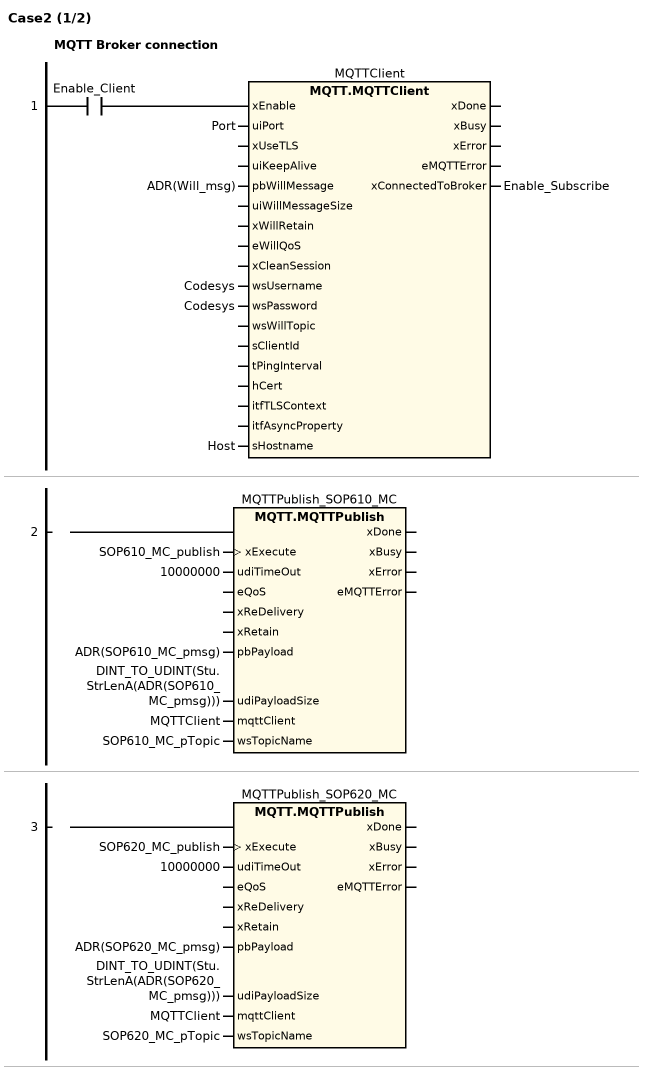
// NETWORK 1: MQTT Broker connection
MQTTClient(
    xEnable := Enable_Client,
    uiPort := Port,
    pbWillMessage := ADR(Will_msg),
    wsUsername := Codesys,
    wsPassword := Codesys,
    sHostname := Host,
    xConnectedToBroker => Enable_Subscribe); // MQTT.MQTTClient

// NETWORK 2
_rt1(CLK := SOP610_MC_publish);
MQTTPublish_SOP610_MC(
    xExecute := _rt1.Q,
    udiTimeOut := 10000000,
    pbPayload := ADR(SOP610_MC_pmsg),
    udiPayloadSize := DINT_TO_UDINT(Stu.StrLenA(ADR(SOP610_MC_pmsg))),
    mqttClient := MQTTClient,
    wsTopicName := SOP610_MC_pTopic); // MQTT.MQTTPublish

// NETWORK 3
_rt2(CLK := SOP620_MC_publish);
MQTTPublish_SOP620_MC(
    xExecute := _rt2.Q,
    udiTimeOut := 10000000,
    pbPayload := ADR(SOP620_MC_pmsg),
    udiPayloadSize := DINT_TO_UDINT(Stu.StrLenA(ADR(SOP620_MC_pmsg))),
    mqttClient := MQTTClient,
    wsTopicName := SOP620_MC_pTopic); // MQTT.MQTTPublish

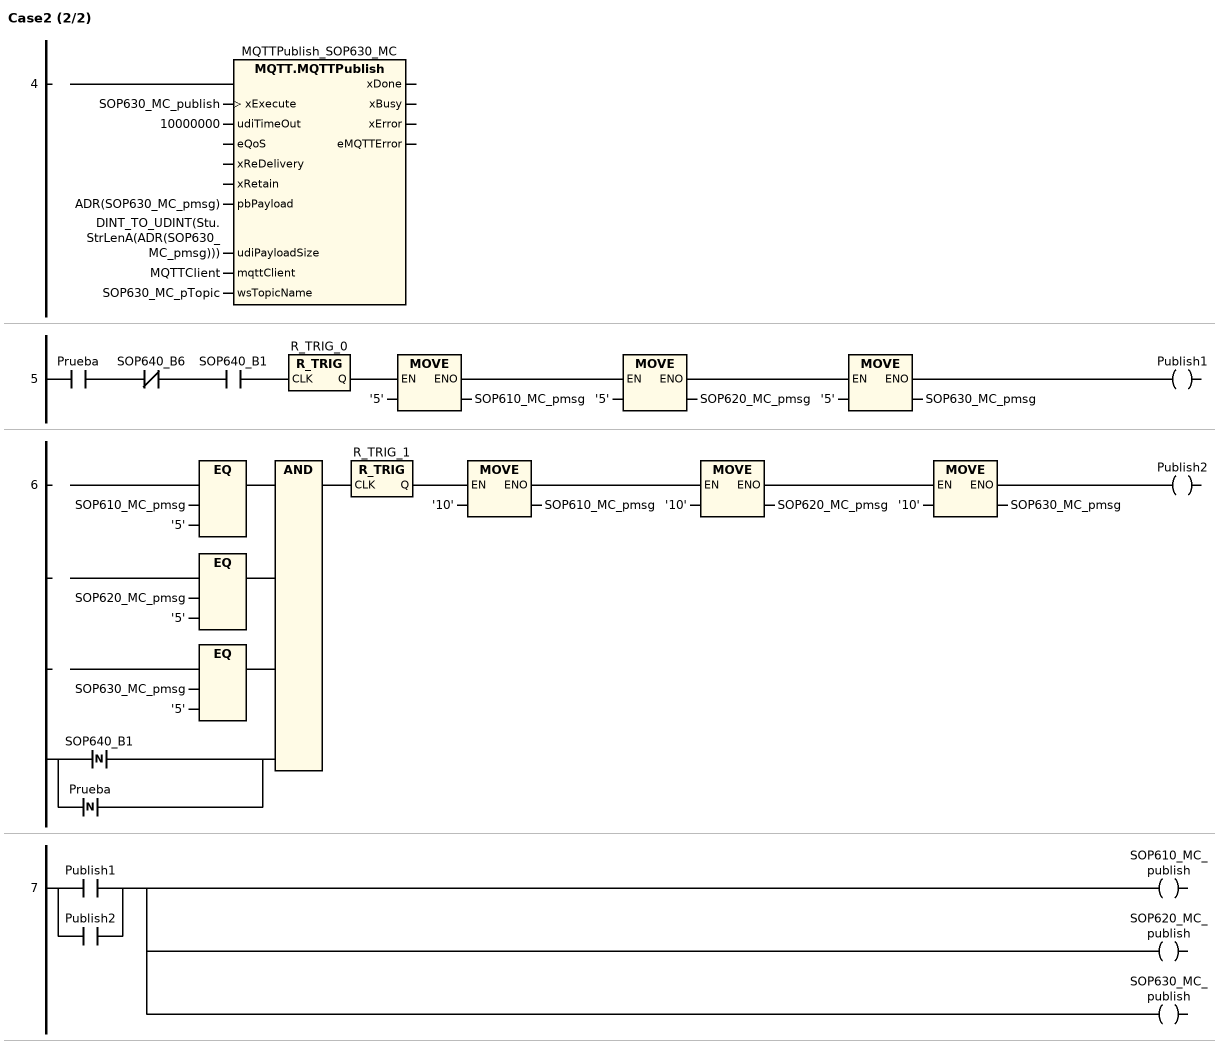
// NETWORK 4
_rt3(CLK := SOP630_MC_publish);
MQTTPublish_SOP630_MC(
    xExecute := _rt3.Q,
    udiTimeOut := 10000000,
    pbPayload := ADR(SOP630_MC_pmsg),
    udiPayloadSize := DINT_TO_UDINT(Stu.StrLenA(ADR(SOP630_MC_pmsg))),
    mqttClient := MQTTClient,
    wsTopicName := SOP630_MC_pTopic); // MQTT.MQTTPublish

// NETWORK 5
R_TRIG_0(CLK := Prueba AND NOT SOP640_B6 AND SOP640_B1); // R_TRIG
_w1 := R_TRIG_0.Q;
IF _w1 THEN SOP610_MC_pmsg := '5'; END_IF
IF _w1 THEN SOP620_MC_pmsg := '5'; END_IF
IF _w1 THEN SOP630_MC_pmsg := '5'; END_IF
Publish1 := _w1;

// NETWORK 6
_ft1(CLK := SOP640_B1);
_ft2(CLK := Prueba);
R_TRIG_1(CLK := SOP610_MC_pmsg = '5' AND SOP620_MC_pmsg = '5' AND SOP630_MC_pmsg = '5' AND (_ft1.Q OR _ft2.Q)); // R_TRIG
_w2 := R_TRIG_1.Q;
IF _w2 THEN SOP610_MC_pmsg := '10'; END_IF
IF _w2 THEN SOP620_MC_pmsg := '10'; END_IF
IF _w2 THEN SOP630_MC_pmsg := '10'; END_IF
Publish2 := _w2;

// NETWORK 7
_w3 := Publish1 OR Publish2;
SOP610_MC_publish := _w3;
SOP620_MC_publish := _w3;
SOP630_MC_publish := _w3;

END_PROGRAM

// Device/Application/Cases/Cases3_4_5
PROGRAM Cases3_4_5
VAR
	MQTTClient: MQTT.MQTTClient; 										// MQTTClient FB
	Port: UINT := 1883; 												// Port
	Will_msg: STRING(1024) := ''; 										// Message if there is disconnection
	Host: STRING(255) := '192.168.1.123'; 								// Broker IP 192.168.1.123 Simumatik
	Codesys: WSTRING(1024) := "codesys";								// Username and password "Codesys"
	Enable_Client: BOOL := TRUE; 										// Establishes connecting with the MQTT broker
	Enable_Subscribe: BOOL;												// Enables subscription
	
	MQTTPublish_SOP610_MC: MQTT.MQTTPublish;								// MQTTPublish FB
	SOP610_MC_publish: BOOL;
	SOP610_MC_pmsg: STRING(1024);
	SOP610_MC_pTopic: WSTRING(1024) := "OP60/SOP610_MC";	
	MQTTPublish_SOP620_MC: MQTT.MQTTPublish;								// MQTTPublish FB
	SOP620_MC_publish: BOOL;
	SOP620_MC_pmsg: STRING(1024);
	SOP620_MC_pTopic: WSTRING(1024) := "OP60/SOP620_MC";
	MQTTPublish_SOP630_MC: MQTT.MQTTPublish;								// MQTTPublish FB
	SOP630_MC_publish: BOOL;
	SOP630_MC_pmsg: STRING(1024);
	SOP630_MC_pTopic: WSTRING(1024) := "OP60/SOP630_MC";
	MQTTPublish_SOP640_MC: MQTT.MQTTPublish;								// MQTTPublish FB
	SOP640_MC_publish: BOOL;
	SOP640_MC_pmsg: STRING(1024);
	SOP640_MC_pTopic: WSTRING(1024) := "OP60/SOP640_MC";
	MQTTPublish_SOP650_MC: MQTT.MQTTPublish;								// MQTTPublish FB
	SOP650_MC_publish: BOOL;
	SOP650_MC_pmsg: STRING(1024);
	SOP650_MC_pTopic: WSTRING(1024) := "OP60/SOP650_MC";
	MQTTPublish_SOP660_MC: MQTT.MQTTPublish;								// MQTTPublish FB
	SOP660_MC_publish: BOOL;
	SOP660_MC_pmsg: STRING(1024);
	SOP660_MC_pTopic: WSTRING(1024) := "OP60/SOP660_MC";
	MQTTPublish_SOP670_MC: MQTT.MQTTPublish;								// MQTTPublish FB
	SOP670_MC_publish: BOOL;
	SOP670_MC_pmsg: STRING(1024);
	SOP670_MC_pTopic: WSTRING(1024) := "OP60/SOP670_MC";
	MQTTPublish_SOP680_MC: MQTT.MQTTPublish;								// MQTTPublish FB
	SOP680_MC_publish: BOOL;
	SOP680_MC_pmsg: STRING(1024);
	SOP680_MC_pTopic: WSTRING(1024) := "OP60/SOP680_MC";
	
	MQTTSubscribe_MC: MQTT.MQTTSubscribe;
	Subscribe_Topic: WSTRING(1024) := "OP60/MC";
	Subscribe_msg: STRING(1024);
	Subscribe_msg_received: BOOL;
	
	R_TRIG_0: R_TRIG;
	R_TRIG_1: R_TRIG;
	R_TRIG_2: R_TRIG;
	R_TRIG_3: R_TRIG;
	R_TRIG_4: R_TRIG;
	R_TRIG_5: R_TRIG;
	R_TRIG_6: R_TRIG;
	R_TRIG_7: R_TRIG;
	R_TRIG_8: R_TRIG;
	Iniciate_publish: BOOL;
	TON_0: TON;
END_VAR
VAR_INPUT
	iSOP610_MC: BOOL;
	iSOP620_MC: BOOL;
	iSOP630_MC: BOOL;
	iSOP640_MC: BOOL;
	iSOP650_MC: BOOL;
	iSOP660_MC: BOOL;
	iSOP670_MC: BOOL;
	iSOP680_MC: BOOL;
END_VAR
VAR // added by the converter: edge detectors and wires of the graphical bodies
    _rt1, _rt2, _rt3, _rt4, _rt5, _rt6, _rt7, _rt8 : R_TRIG;
    _w1, _w2, _w3, _w4, _w5, _w6, _w7, _w8, _w9 : BOOL;
END_VAR

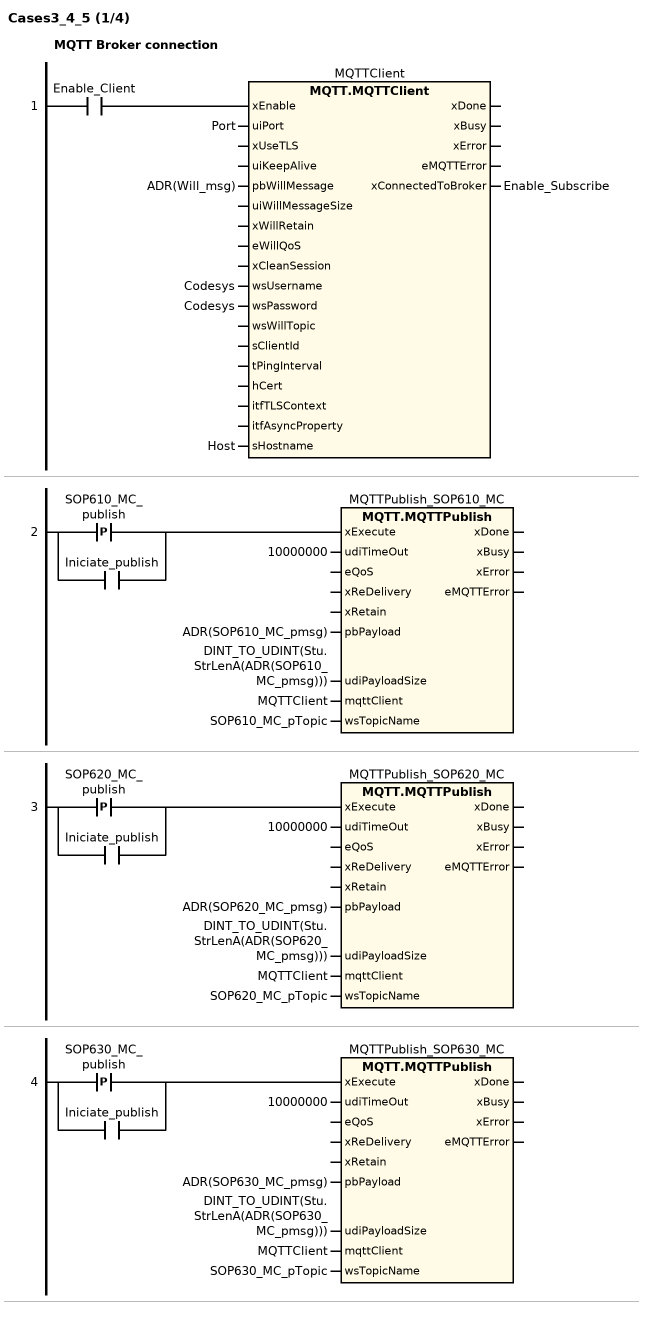
// NETWORK 1: MQTT Broker connection
MQTTClient(
    xEnable := Enable_Client,
    uiPort := Port,
    pbWillMessage := ADR(Will_msg),
    wsUsername := Codesys,
    wsPassword := Codesys,
    sHostname := Host,
    xConnectedToBroker => Enable_Subscribe); // MQTT.MQTTClient

// NETWORK 2
_rt1(CLK := SOP610_MC_publish);
MQTTPublish_SOP610_MC(
    xExecute := _rt1.Q OR Iniciate_publish,
    udiTimeOut := 10000000,
    pbPayload := ADR(SOP610_MC_pmsg),
    udiPayloadSize := DINT_TO_UDINT(Stu.StrLenA(ADR(SOP610_MC_pmsg))),
    mqttClient := MQTTClient,
    wsTopicName := SOP610_MC_pTopic); // MQTT.MQTTPublish

// NETWORK 3
_rt2(CLK := SOP620_MC_publish);
MQTTPublish_SOP620_MC(
    xExecute := _rt2.Q OR Iniciate_publish,
    udiTimeOut := 10000000,
    pbPayload := ADR(SOP620_MC_pmsg),
    udiPayloadSize := DINT_TO_UDINT(Stu.StrLenA(ADR(SOP620_MC_pmsg))),
    mqttClient := MQTTClient,
    wsTopicName := SOP620_MC_pTopic); // MQTT.MQTTPublish

// NETWORK 4
_rt3(CLK := SOP630_MC_publish);
MQTTPublish_SOP630_MC(
    xExecute := _rt3.Q OR Iniciate_publish,
    udiTimeOut := 10000000,
    pbPayload := ADR(SOP630_MC_pmsg),
    udiPayloadSize := DINT_TO_UDINT(Stu.StrLenA(ADR(SOP630_MC_pmsg))),
    mqttClient := MQTTClient,
    wsTopicName := SOP630_MC_pTopic); // MQTT.MQTTPublish

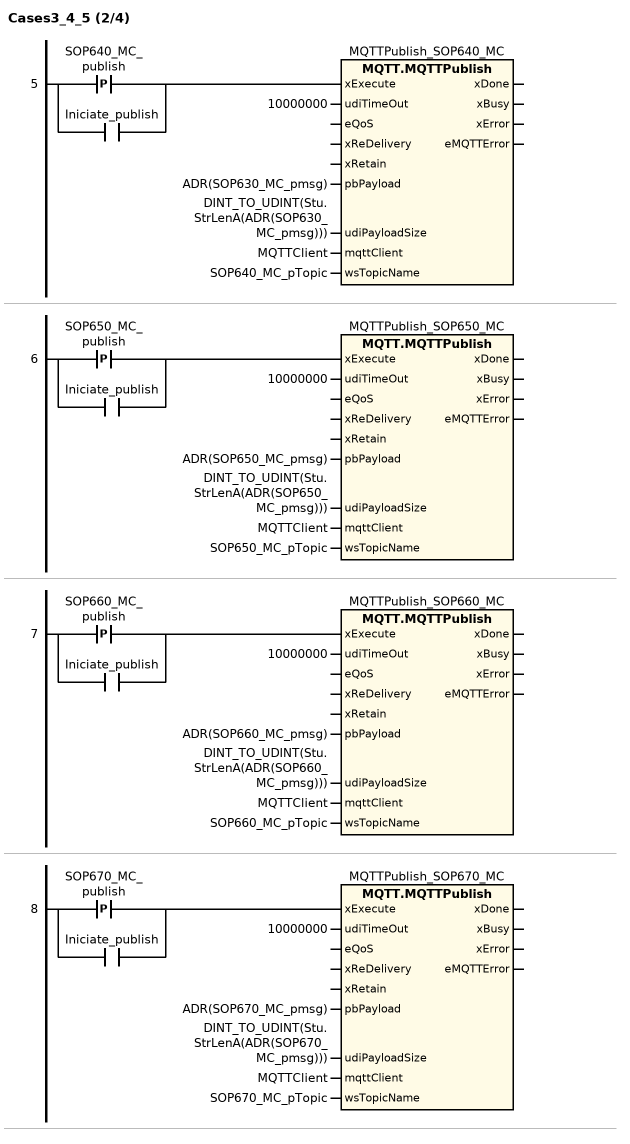
// NETWORK 5
_rt4(CLK := SOP640_MC_publish);
MQTTPublish_SOP640_MC(
    xExecute := _rt4.Q OR Iniciate_publish,
    udiTimeOut := 10000000,
    pbPayload := ADR(SOP630_MC_pmsg),
    udiPayloadSize := DINT_TO_UDINT(Stu.StrLenA(ADR(SOP630_MC_pmsg))),
    mqttClient := MQTTClient,
    wsTopicName := SOP640_MC_pTopic); // MQTT.MQTTPublish

// NETWORK 6
_rt5(CLK := SOP650_MC_publish);
MQTTPublish_SOP650_MC(
    xExecute := _rt5.Q OR Iniciate_publish,
    udiTimeOut := 10000000,
    pbPayload := ADR(SOP650_MC_pmsg),
    udiPayloadSize := DINT_TO_UDINT(Stu.StrLenA(ADR(SOP650_MC_pmsg))),
    mqttClient := MQTTClient,
    wsTopicName := SOP650_MC_pTopic); // MQTT.MQTTPublish

// NETWORK 7
_rt6(CLK := SOP660_MC_publish);
MQTTPublish_SOP660_MC(
    xExecute := _rt6.Q OR Iniciate_publish,
    udiTimeOut := 10000000,
    pbPayload := ADR(SOP660_MC_pmsg),
    udiPayloadSize := DINT_TO_UDINT(Stu.StrLenA(ADR(SOP660_MC_pmsg))),
    mqttClient := MQTTClient,
    wsTopicName := SOP660_MC_pTopic); // MQTT.MQTTPublish

// NETWORK 8
_rt7(CLK := SOP670_MC_publish);
MQTTPublish_SOP670_MC(
    xExecute := _rt7.Q OR Iniciate_publish,
    udiTimeOut := 10000000,
    pbPayload := ADR(SOP670_MC_pmsg),
    udiPayloadSize := DINT_TO_UDINT(Stu.StrLenA(ADR(SOP670_MC_pmsg))),
    mqttClient := MQTTClient,
    wsTopicName := SOP670_MC_pTopic); // MQTT.MQTTPublish

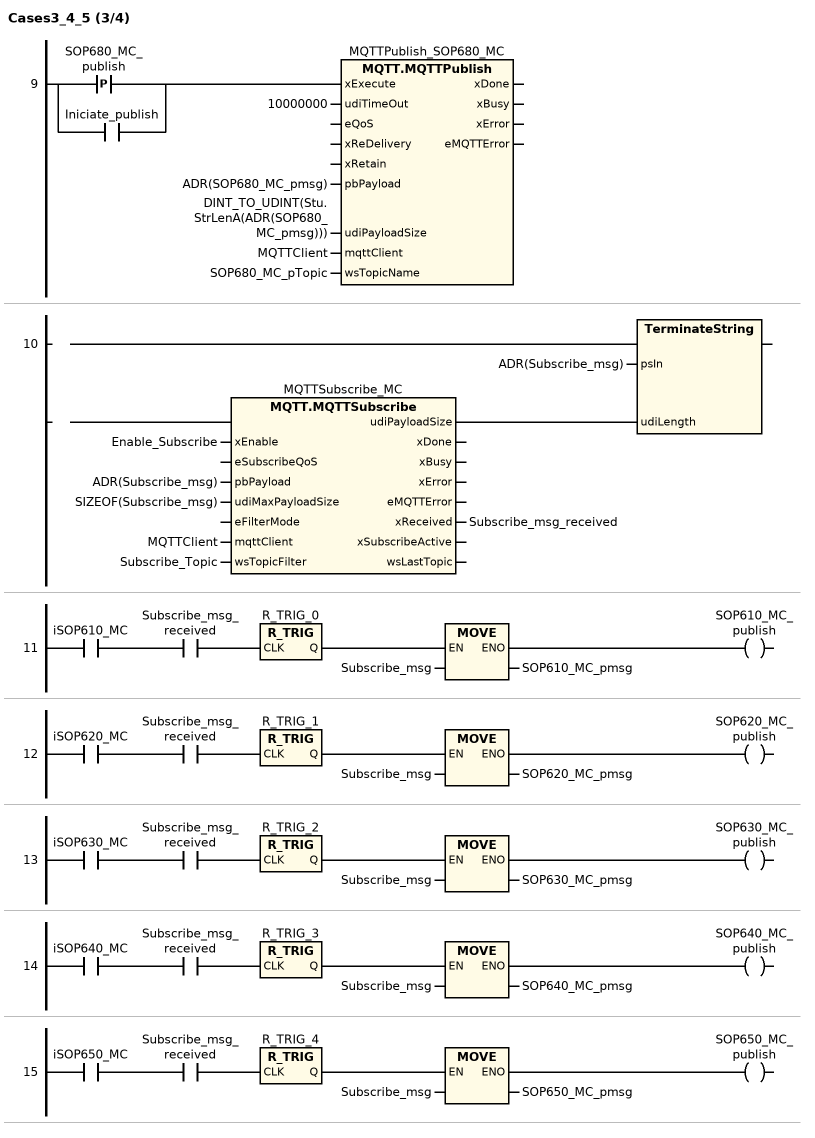
// NETWORK 9
_rt8(CLK := SOP680_MC_publish);
MQTTPublish_SOP680_MC(
    xExecute := _rt8.Q OR Iniciate_publish,
    udiTimeOut := 10000000,
    pbPayload := ADR(SOP680_MC_pmsg),
    udiPayloadSize := DINT_TO_UDINT(Stu.StrLenA(ADR(SOP680_MC_pmsg))),
    mqttClient := MQTTClient,
    wsTopicName := SOP680_MC_pTopic); // MQTT.MQTTPublish

// NETWORK 10
MQTTSubscribe_MC(
    xEnable := Enable_Subscribe,
    pbPayload := ADR(Subscribe_msg),
    udiMaxPayloadSize := SIZEOF(Subscribe_msg),
    mqttClient := MQTTClient,
    wsTopicFilter := Subscribe_Topic,
    xReceived => Subscribe_msg_received); // MQTT.MQTTSubscribe
TerminateString(psIn := ADR(Subscribe_msg), udiLength := MQTTSubscribe_MC.udiPayloadSize);

// NETWORK 11
R_TRIG_0(CLK := iSOP610_MC AND Subscribe_msg_received); // R_TRIG
_w1 := R_TRIG_0.Q;
IF _w1 THEN SOP610_MC_pmsg := Subscribe_msg; END_IF
SOP610_MC_publish := _w1;

// NETWORK 12
R_TRIG_1(CLK := iSOP620_MC AND Subscribe_msg_received); // R_TRIG
_w2 := R_TRIG_1.Q;
IF _w2 THEN SOP620_MC_pmsg := Subscribe_msg; END_IF
SOP620_MC_publish := _w2;

// NETWORK 13
R_TRIG_2(CLK := iSOP630_MC AND Subscribe_msg_received); // R_TRIG
_w3 := R_TRIG_2.Q;
IF _w3 THEN SOP630_MC_pmsg := Subscribe_msg; END_IF
SOP630_MC_publish := _w3;

// NETWORK 14
R_TRIG_3(CLK := iSOP640_MC AND Subscribe_msg_received); // R_TRIG
_w4 := R_TRIG_3.Q;
IF _w4 THEN SOP640_MC_pmsg := Subscribe_msg; END_IF
SOP640_MC_publish := _w4;

// NETWORK 15
R_TRIG_4(CLK := iSOP650_MC AND Subscribe_msg_received); // R_TRIG
_w5 := R_TRIG_4.Q;
IF _w5 THEN SOP650_MC_pmsg := Subscribe_msg; END_IF
SOP650_MC_publish := _w5;

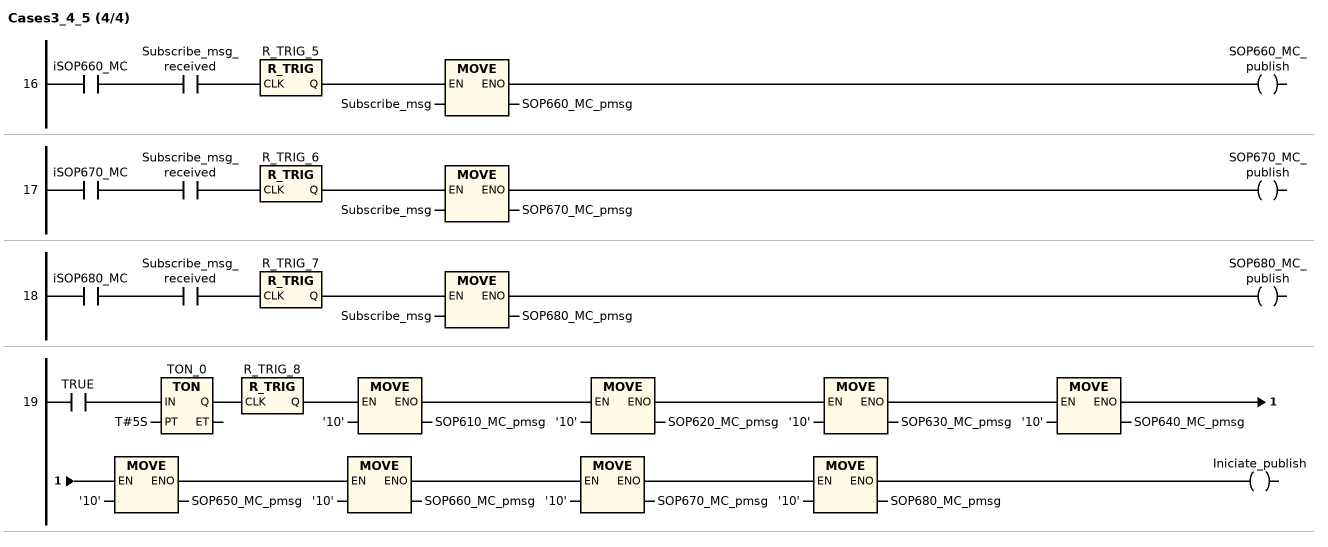
// NETWORK 16
R_TRIG_5(CLK := iSOP660_MC AND Subscribe_msg_received); // R_TRIG
_w6 := R_TRIG_5.Q;
IF _w6 THEN SOP660_MC_pmsg := Subscribe_msg; END_IF
SOP660_MC_publish := _w6;

// NETWORK 17
R_TRIG_6(CLK := iSOP670_MC AND Subscribe_msg_received); // R_TRIG
_w7 := R_TRIG_6.Q;
IF _w7 THEN SOP670_MC_pmsg := Subscribe_msg; END_IF
SOP670_MC_publish := _w7;

// NETWORK 18
R_TRIG_7(CLK := iSOP680_MC AND Subscribe_msg_received); // R_TRIG
_w8 := R_TRIG_7.Q;
IF _w8 THEN SOP680_MC_pmsg := Subscribe_msg; END_IF
SOP680_MC_publish := _w8;

// NETWORK 19
TON_0(IN := TRUE, PT := T#5S); // TON
R_TRIG_8(CLK := TON_0.Q); // R_TRIG
_w9 := R_TRIG_8.Q;
IF _w9 THEN SOP610_MC_pmsg := '10'; END_IF
IF _w9 THEN SOP620_MC_pmsg := '10'; END_IF
IF _w9 THEN SOP630_MC_pmsg := '10'; END_IF
IF _w9 THEN SOP640_MC_pmsg := '10'; END_IF
IF _w9 THEN SOP650_MC_pmsg := '10'; END_IF
IF _w9 THEN SOP660_MC_pmsg := '10'; END_IF
IF _w9 THEN SOP670_MC_pmsg := '10'; END_IF
IF _w9 THEN SOP680_MC_pmsg := '10'; END_IF
Iniciate_publish := _w9;

END_PROGRAM

// Device/Application/MQTTSub
PROGRAM MQTTSub
VAR
	//Define Client
	MQTTCLient5 : MQTT.MQTTClient;		
	MQTTReady: BOOL;								
	Enable_Client : BOOL := TRUE;										
	Port : UINT := 1883;
	Will_msg: STRING(1024) := ''; 										// Message if there is disconnection
	Host: STRING(255) := '192.168.1.123'; 								// Broker IP 192.168.1.123 Simumatik
	Codesys: WSTRING(1024) := "codesys";
	
	// Define Subscriber
	MQTTSubscriber: MQTT.MQTTSubscribe;
	Enable_Subscribe: BOOL;
	Received_messages: ARRAY [1..3] OF STRING(1024) := ['', '', ''];	// Received messages
	New_message: ARRAY [1..3] OF BOOL;									// This is done to avoid errors
	Topics: ARRAY [1..3] OF WSTRING(1024) := ["Subscriber1","Subscriber2","Subscriber3"];
	
	i: DINT := 1;
	Delay: TON;
	DelayTime: TIME;
END_VAR

MQTTClient5(xEnable:=Enable_Client, uiPort:=Port, pbWillMessage:=ADR(Will_msg), wsUsername:=Codesys, wsPassword:=Codesys, sHostname:=Host, xConnectedToBroker => MQTTReady);  // Define Client

IF MQTTReady THEN
	MQTTSubscriber(xEnable:= TRUE, pbPayload:= ADR(Received_messages[i]), udiMaxPayloadSize:= SIZEOF(Received_messages[i]), mqttClient:= MQTTClient5, wsTopicFilter:= Topics[i], xReceived => New_message[i]);
	Delay(IN:=TRUE, PT:=T#100MS, ET => DelayTime);
	IF NOT(Delay.Q) THEN
		RETURN;
	END_IF
	Delay(IN:=FALSE);
	MQTTSubscriber(xEnable:= FALSE, pbPayload:= ADR(Received_messages[i]), udiMaxPayloadSize:= SIZEOF(Received_messages[i]), mqttClient:= MQTTClient5, wsTopicFilter:= Topics[i], xReceived => New_message[i]);
END_IF

IF i = (UPPER_BOUND(Received_messages,1)) THEN
	i := LOWER_BOUND(Received_messages,1)-1;
END_IF
i := i+1;

END_PROGRAM

// Device/Application/FBs/EraseSeconds
FUNCTION EraseSeconds : STRING // Returns TIME STRING in HH:MM:SS to HH:MM format 
VAR_INPUT
	iTime_hh_mm_ss: STRING;
END_VAR
VAR
END_VAR

EraseSeconds := LEFT(iTime_hh_mm_ss,5);

END_FUNCTION

// Device/Application/Pruebas
PROGRAM Pruebas
VAR

	Output: SysFile.RTS_IEC_HANDLE;
	TON_0: TON;
	TimerON: BOOL;
	TimerON_0: TIME;
	Salida: __XWORD;
	pbyBuffer: POINTER TO BYTE := 4096;
	ulSize: __XWORD := 4096;
	pResult: POINTER TO SysFile.RTS_IEC_RESULT;
	szFile: REFERENCE TO STRING;
END_VAR

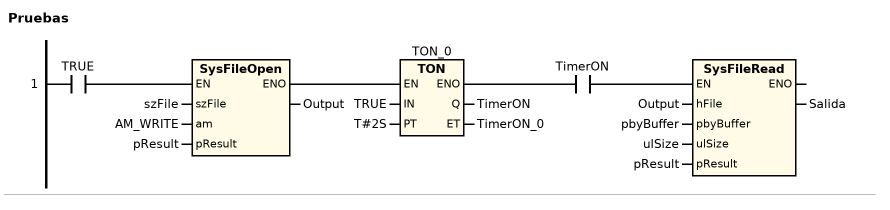
// NETWORK 1
Output := SysFileOpen(szFile := szFile, am := AM_WRITE, pResult := pResult);
TON_0(IN := TRUE, PT := T#2S, Q => TimerON, ET => TimerON_0); // TON
IF TRUE AND TimerON THEN
    Salida := SysFileRead(hFile := Output, pbyBuffer := pbyBuffer, ulSize := ulSize, pResult := pResult);
END_IF

END_PROGRAM

// Device/Application/MQTTPub
PROGRAM MQTTPub
VAR
	//Define Client
	MQTTCLient4 : MQTT.MQTTClient;										
	Enable_Client : BOOL := TRUE;										
	Port : UINT := 1883;
	Will_msg: STRING(1024) := ''; 										// Message if there is disconnection
	Host: STRING(255) := '192.168.1.123'; 								// Broker IP 192.168.1.123 Simumatik
	Codesys: WSTRING(1024) := "codesys";
	Enable_Publish: BOOL;												// Rising edge activates Publisher FB
	
	//Define Publisher
	MQTTPublisher: MQTT.MQTTPublish;
	Topics: ARRAY [1..3] OF WSTRING(1024) := ["Publish","Publish2","Publish3"];	// All the topics
	Publish_msg: ARRAY [1..3] OF STRING(1024);			// Messages to publish
	Publish_last_msg: ARRAY [1..3] OF STRING(1024);		// Last messages to publish

	i : DINT := 1; 		//index
	Delay: TON;			// Timer to delay
END_VAR

MQTTClient4(xEnable:=Enable_Client, uiPort:=Port, pbWillMessage:=ADR(Will_msg), wsUsername:=Codesys, wsPassword:=Codesys, sHostname:=Host,);  // Define Client

// Publish the messages that have change
IF NOT (Publish_msg[i] = Publish_last_msg[i]) THEN
	Enable_Publish:= TRUE;
	MQTTPublisher(xExecute:=Enable_Publish, udiTimeOut:=1000000, pbPayload:=ADR(Publish_msg[i]), udiPayloadSize:=DINT_TO_UDINT(Stu.StrLenA(ADR(Publish_msg[i]))), mqttclient:=MQTTClient4, wsTopicName:=Topics[i]);
	// Delay 50miliseconds;
	Delay(IN:=TRUE, PT:=T#50MS);
	IF NOT(Delay.Q) THEN
   		RETURN;
	END_IF
	Delay(IN:=FALSE);
	Enable_Publish:= FALSE;
	MQTTPublisher(xExecute:=FALSE, udiTimeOut:=1000000, pbPayload:=ADR(Publish_msg[i]), udiPayloadSize:=DINT_TO_UDINT(Stu.StrLenA(ADR(Publish_msg[i]))), mqttclient:=MQTTClient4, wsTopicName:=Topics[i]);
	// To avoid missing messages
	//MQTTPublisher(xExecute:=TRUE, udiTimeOut:=1000000, pbPayload:=ADR(Publish_msg[i]), udiPayloadSize:=DINT_TO_UDINT(Stu.StrLenA(ADR(Publish_msg[i]))), mqttclient:=MQTTClient4, wsTopicName:=Topics[i]);
	//MQTTPublisher(xExecute:=FALSE, udiTimeOut:=1000000, pbPayload:=ADR(Publish_msg[i]), udiPayloadSize:=DINT_TO_UDINT(Stu.StrLenA(ADR(Publish_msg[i]))), mqttclient:=MQTTClient4, wsTopicName:=Topics[i]);
	
	Publish_last_msg[i] := Publish_msg[i];
	
END_IF

// IF Enable_Publish = TRUE THEN
// 	// Delay 50miliseconds;
// 	Delay(IN:=TRUE, PT:=T#50MS);
// 	IF NOT(Delay.Q) THEN
//    		RETURN;
// 	END_IF
// 	Delay(IN:=FALSE);
// 	Enable_Publish:= FALSE;
// 	MQTTPublisher(xExecute:=Enable_Publish);
// END_IF


// Control the index
IF i = (UPPER_BOUND(Publish_msg,1)) THEN
	i := LOWER_BOUND(Publish_msg,1)-1;
END_IF
i := i+1;

END_PROGRAM

// Device/Application/Production
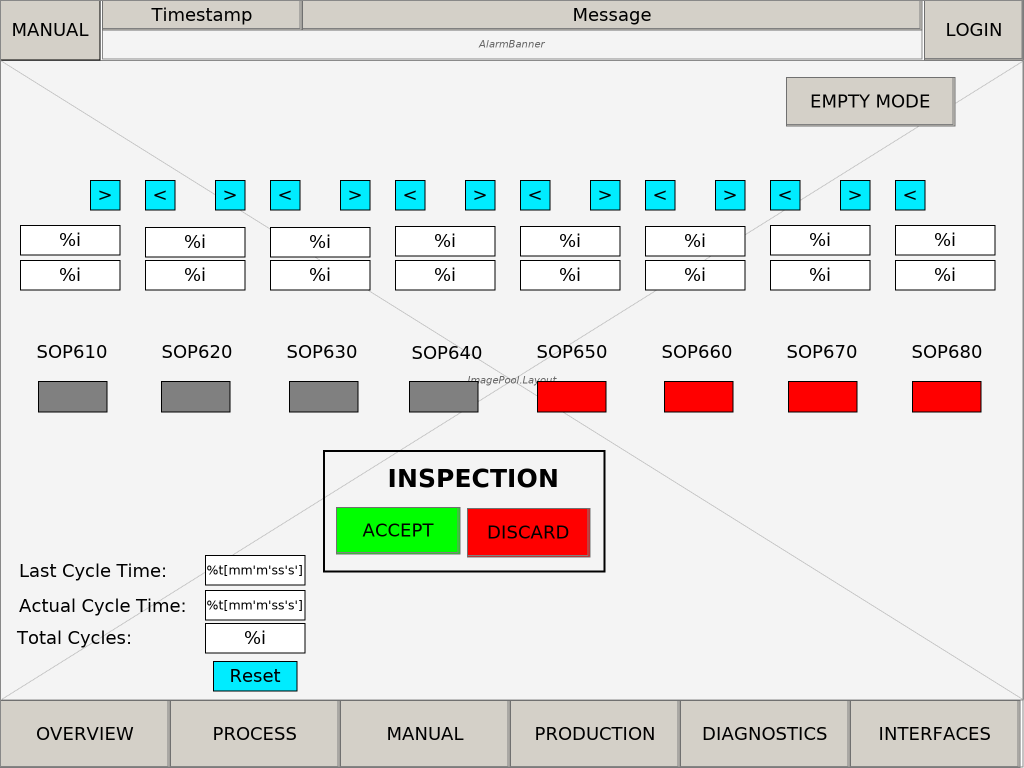
VISUALIZATION Production  // 1024x768, background image ImagePool.Layout
    Image (0,60 1024x640), image: ImagePool.Layout
    Rectangle (0,0 100x60), "AUTO"
    Rectangle (0,0 100x60), "MANUAL", invisible if: OP60_Auto
    AlarmBanner (102,29 820x30)
        p1521930926: __All
        p1663851261: __All
    Button (924,0 100x60), "LOGIN"
    Button (102,0 200x30), "Timestamp"
    Button (302,0 620x30), "Message"
    Label (145,337 104x30), "SOP620"
    Label (20,337 104x30), "SOP610"
    Label (270,337 104x30), "SOP630"
    Label (395,338 104x30), "SOP640"
    Label (520,337 104x30), "SOP650"
    Label (645,337 104x30), "SOP660"
    Label (895,337 104x30), "SOP680"
    Label (770,337 104x30), "SOP670"
    Rectangle (20,260 100x30), "%i", text variable: SOP610_PD.ProductNr
    Rectangle (20,225 100x30), "%i", text variable: SOP610_PD.IDNumber
    Rectangle (145,227 100x30), "%i", text variable: SOP620_PD.IDNumber
    Rectangle (145,260 100x30), "%i", text variable: SOP620_PD.ProductNr
    Rectangle (270,227 100x30), "%i", text variable: SOP630_PD.IDNumber
    Rectangle (270,260 100x30), "%i", text variable: SOP630_PD.ProductNr
    Rectangle (395,226 100x30), "%i", text variable: SOP640_PD.IDNumber
    Rectangle (395,260 100x30), "%i", text variable: SOP640_PD.ProductNr
    Rectangle (520,226 100x30), "%i", text variable: SOP650_PD.IDNumber
    Rectangle (520,260 100x30), "%i", text variable: SOP650_PD.ProductNr
    Rectangle (645,226 100x30), "%i", text variable: SOP660_PD.IDNumber
    Rectangle (645,260 100x30), "%i", text variable: SOP660_PD.ProductNr
    Rectangle (770,225 100x30), "%i", text variable: SOP670_PD.IDNumber
    Rectangle (770,260 100x30), "%i", text variable: SOP670_PD.ProductNr
    Rectangle (895,225 100x30), "%i", text variable: SOP680_PD.IDNumber
    Rectangle (895,260 100x30), "%i", text variable: SOP680_PD.ProductNr
    Group (323,450 282x122), invisible if: not HMI_SOP640_Inspecting
        Rectangle (0,0 282x122)
        Button (13,57 124x47), "ACCEPT"
            tap HMI_SOP640_Accept
        Label (39,13 223x30), "INSPECTION"
        Button (144,58 123x49), "DISCARD"
            tap HMI_SOP640_Discard
    Group (0,700 1020x68)
        Button (0,0 170x68), "OVERVIEW"
            toggle OP60_Visu.CV_Overview
            OnMouseDown:  Assign=Overview, Type=Assignment
        Button (170,0 170x68), "PROCESS"
            toggle OP60_Visu.CV_Process
            OnMouseDown:  Assign=Process, Type=Assignment
        Button (340,0 170x68), "MANUAL"
            toggle OP60_Visu.CV_Manual_SOP610t630
            OnMouseDown:  Assign=Manual_SOP610t630, Type=Assignment
        Button (510,0 170x68), "PRODUCTION"
            toggle OP60_Visu.CV_Production
            OnMouseDown:  Assign=Production, Type=Assignment
        Button (680,0 170x68), "DIAGNOSTICS"
            toggle OP60_Visu.CV_Diagnostics
            OnMouseDown:  Assign=Diagnostics, Type=Assignment
        Button (850,0 170x68), "INTERFACES"
            toggle OP60_Visu.CV_Interfaces
            OnMouseDown:  Assign=Interfaces, Type=Assignment
    Rectangle (90,180 30x30), ">"
        tap HMI_SOP610_ManPDFwd
    Rectangle (215,180 30x30), ">"
        tap HMI_SOP620_ManPDFwd
    Rectangle (145,180 30x30), "<"
        tap HMI_SOP620_ManPDRev
    Rectangle (340,180 30x30), ">"
        tap HMI_SOP630_ManPDFwd
    Rectangle (270,180 30x30), "<"
        tap HMI_SOP630_ManPDRev
    Rectangle (465,180 30x30), ">"
        tap HMI_SOP640_ManPDFwd
    Rectangle (395,180 30x30), "<"
        tap HMI_SOP640_ManPDRev
    Rectangle (590,180 30x30), ">"
        tap HMI_SOP650_ManPDFwd
    Rectangle (520,180 30x30), "<"
        tap HMI_SOP650_ManPDRev
    Rectangle (715,180 30x30), ">"
        tap HMI_SOP660_ManPDFwd
    Rectangle (645,180 30x30), "<"
        tap HMI_SOP660_ManPDRev
    Rectangle (840,180 30x30), ">"
        tap HMI_SOP670_ManPDFwd
    Rectangle (770,180 30x30), "<"
        tap HMI_SOP670_ManPDRev
    Rectangle (895,180 30x30), "<"
        tap HMI_SOP680_ManPDRev
    Label (16,591 193x30), "Actual Cycle Time:"
    Label (14,623 193x30), "Total Cycles:"
    Rectangle (213,661 84x30), "Reset"
        tap HMI_TotalCyclesReset
    Rectangle (205,590 100x30), "%t[mm'm'ss's']", text variable: OP60_ActualCycleTime
    Rectangle (205,623 100x30), "%i", text variable: OP60_TotalCycles
    Button (786,77 169x49), "EMPTY MODE"
        toggle GVL.OP60_EmptyMode
    Group (38,381 943x31)
        Rectangle (371,0 69x31), invisible if: not STRING_TO_BOOL(SOP640_B1_msg)
        Rectangle (251,0 69x31), invisible if: not STRING_TO_BOOL(SOP630_B1_msg)
        Rectangle (123,0 69x31), invisible if: not STRING_TO_BOOL(SOP620_B1_msg)
        Rectangle (0,0 69x31), invisible if: not STRING_TO_BOOL(SOP610_B1_msg)
        Rectangle (499,0 69x31), invisible if: not STRING_TO_BOOL(SOP650_B1_msg)
            toggle SOP650_PD.Status.6
        Rectangle (626,0 69x31), invisible if: not STRING_TO_BOOL(SOP660_B1_msg)
            toggle SOP660_PD.Status.6
        Rectangle (750,0 69x31), invisible if: not STRING_TO_BOOL(SOP670_B1_msg)
            toggle SOP670_PD.Status.6
        Rectangle (874,0 69x31), invisible if: not STRING_TO_BOOL(SOP680_B1_msg)
            toggle SOP680_PD.Status.6
    Label (16,556 193x30), "Last Cycle Time:"
    Rectangle (205,555 100x30), "%t[mm'm'ss's']", text variable: OP60_LastCycleTime
END_VISUALIZATION

// /Diagnostics
VISUALIZATION Diagnostics  // 1024x768
END_VISUALIZATION

// Device/Application/Overview
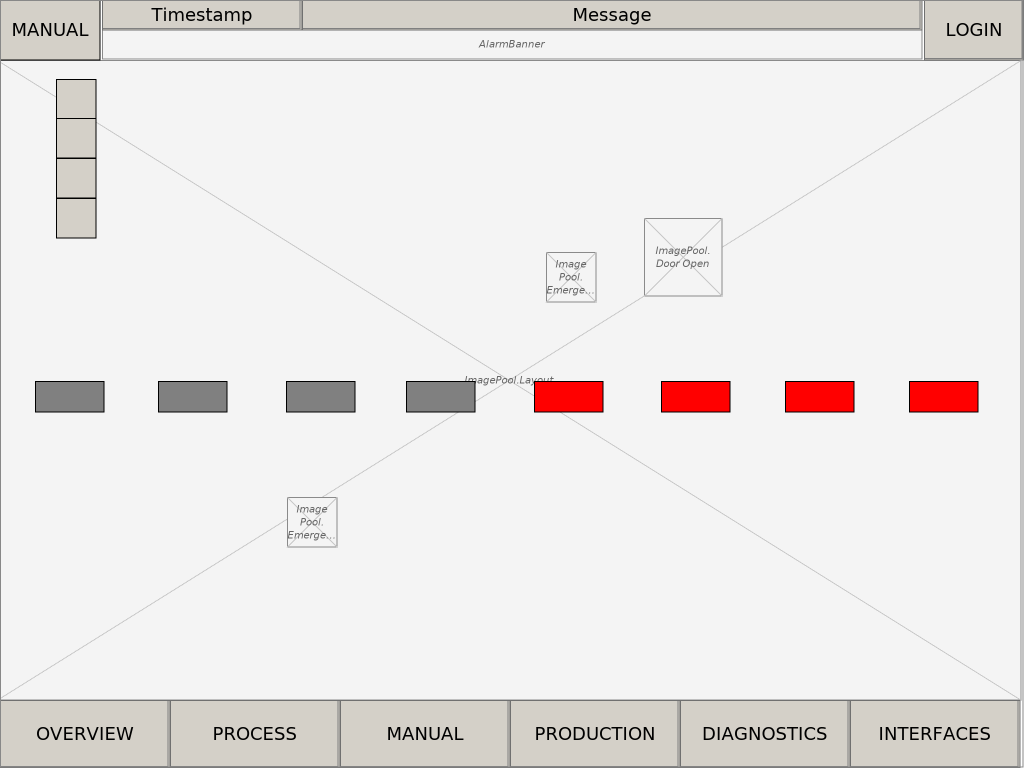
VISUALIZATION Overview  // 1024x768
    Image (-3,60 1024x640), image: ImagePool.Layout
    Rectangle (0,0 100x60), "AUTO"
    Rectangle (0,0 100x60), "MANUAL", invisible if: OP60_Auto
    AlarmBanner (102,29 820x30)
        p1521930926: __All
        p1663851261: __All
    Button (924,0 100x60), "LOGIN"
    Button (102,0 200x30), "Timestamp"
    Button (302,0 620x30), "Message"
    Group (56,79 40x159)
        Rectangle (0,0 40x40)
            toggle SOP600_H9
        Rectangle (0,39 40x40)
            toggle SOP600_H8
        Rectangle (0,79 40x40)
            toggle SOP600_H7
        Rectangle (0,119 40x40)
            toggle SOP600_H6
    Image (287,497 50x50), invisible if: SOP600_NS1, image: ImagePool.Emergency Stop
    Image (546,252 50x50), invisible if: SOP690_NS1, image: ImagePool.Emergency Stop
    Image (644,218 78x78), invisible if: SOP690_B1, image: ImagePool.Door Open
    Group (0,700 1020x68)
        Button (0,0 170x68), "OVERVIEW"
            toggle OP60_Visu.CV_Overview
            OnMouseDown:  Assign=Overview, Type=Assignment
        Button (170,0 170x68), "PROCESS"
            toggle OP60_Visu.CV_Process
            OnMouseDown:  Assign=Process, Type=Assignment
        Button (340,0 170x68), "MANUAL"
            toggle OP60_Visu.CV_Manual_SOP610t630
            OnMouseDown:  Assign=Manual_SOP610t630, Type=Assignment
        Button (510,0 170x68), "PRODUCTION"
            toggle OP60_Visu.CV_Production
            OnMouseDown:  Assign=Production, Type=Assignment
        Button (680,0 170x68), "DIAGNOSTICS"
            toggle OP60_Visu.CV_Diagnostics
            OnMouseDown:  Assign=Diagnostics, Type=Assignment
        Button (850,0 170x68), "INTERFACES"
            toggle OP60_Visu.CV_Interfaces
            OnMouseDown:  Assign=Interfaces, Type=Assignment
    Group (35,381 943x31)
        Rectangle (371,0 69x31), invisible if: not STRING_TO_BOOL(SOP640_B1_msg)
        Rectangle (251,0 69x31), invisible if: not STRING_TO_BOOL(SOP630_B1_msg)
        Rectangle (123,0 69x31), invisible if: not STRING_TO_BOOL(SOP620_B1_msg)
        Rectangle (0,0 69x31), invisible if: not STRING_TO_BOOL(SOP610_B1_msg)
        Rectangle (499,0 69x31), invisible if: not STRING_TO_BOOL(SOP650_B1_msg)
            toggle SOP650_PD.Status.6
        Rectangle (626,0 69x31), invisible if: not STRING_TO_BOOL(SOP660_B1_msg)
            toggle SOP660_PD.Status.6
        Rectangle (750,0 69x31), invisible if: not STRING_TO_BOOL(SOP670_B1_msg)
            toggle SOP670_PD.Status.6
        Rectangle (874,0 69x31), invisible if: not STRING_TO_BOOL(SOP680_B1_msg)
            toggle SOP680_PD.Status.6
END_VISUALIZATION

// Device/Application/Manual_SOP640
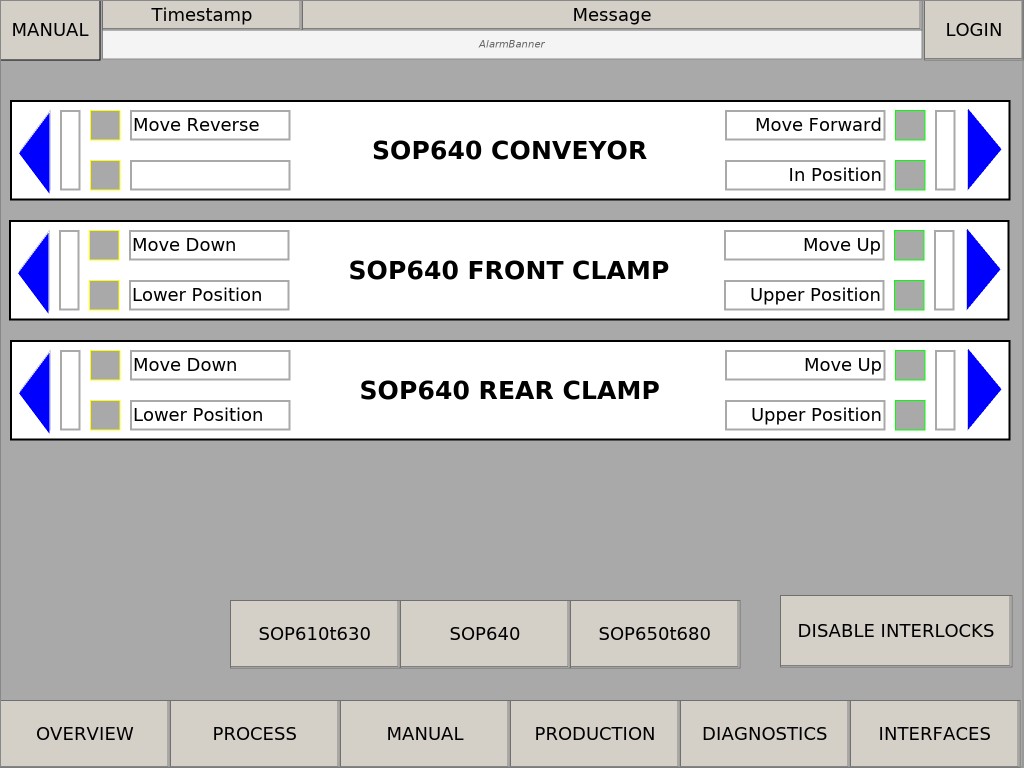
VISUALIZATION Manual_SOP640  // 1024x768
    Rectangle (0,0 100x60), "AUTO"
    Rectangle (0,0 100x60), "MANUAL", invisible if: OP60_Auto
    AlarmBanner (102,29 820x30)
        p1521930926: __All
        p1663851261: __All
    Button (924,0 100x60), "LOGIN"
    Button (102,0 200x30), "Timestamp"
    Button (302,0 620x30), "Message"
    Button (0,700 170x68), "OVERVIEW"
        toggle OP60_Visu.CV_Overview
        OnMouseDown:  Assign=Overview, Type=Assignment
    Button (170,700 170x68), "PROCESS"
        toggle OP60_Visu.CV_Process
        OnMouseDown:  Assign=Process, Type=Assignment
    Button (340,700 170x68), "MANUAL"
        toggle OP60_Visu.CV_Manual_SOP610t630
        OnMouseDown:  Assign=Manual_SOP610t630, Type=Assignment
    Button (510,700 170x68), "PRODUCTION"
        toggle OP60_Visu.CV_Production
        OnMouseDown:  Assign=Production, Type=Assignment
    Button (680,700 170x68), "DIAGNOSTICS"
        toggle OP60_Visu.CV_Diagnostics
        OnMouseDown:  Assign=Diagnostics, Type=Assignment
    Button (850,700 170x68), "INTERFACES"
        toggle OP60_Visu.CV_Interfaces
        OnMouseDown:  Assign=Interfaces, Type=Assignment
    Group (10,100 1000x100)
        Rectangle (0,0 1000x100), "SOP640 CONVEYOR"
        Polygon (10,50) (40,10) (40,90) (10,50) (10,50)
        Rectangle (50,10 20x80)
            toggle HMI_SOP640_ManMoveRev
        Polygon (990,50) (957,10) (957,90) (990,50) (990,50)
        Rectangle (925,10 20x80)
            toggle HMI_SOP640_ManMoveFwd
        Rectangle (715,10 160x30), "Move Forward"
        Rectangle (715,60 160x30), "In Position"
        Rectangle (120,10 160x30), "Move Reverse"
        Rectangle (120,60 160x30), invisible if: TRUE
        Rectangle (885,10 30x30)
            toggle SOP640_KM1
        Rectangle (80,60 30x30), invisible if: TRUE
        Rectangle (80,10 30x30)
            toggle SOP640_KM2
        Rectangle (885,60 30x30)
            toggle SOP640_B1
        Polygon (991,49) (958,9) (958,89) (991,49) (991,49), invisible if: not OP60_Manual
            tap HMI_SOP640_ManMoveFwd
        Polygon (9,53) (39,13) (39,93) (9,53) (9,53), invisible if: not OP60_Manual
            tap HMI_SOP640_ManMoveRev
    Group (9,220 1000x100)
        Rectangle (0,0 1000x100), "SOP640 FRONT CLAMP"
        Polygon (10,50) (40,10) (40,90) (10,50) (10,50)
        Rectangle (50,10 20x80)
            toggle HMI_SOP640_ManFrontDown
        Polygon (990,50) (957,10) (957,90) (990,50) (990,50)
        Rectangle (925,10 20x80)
            toggle HMI_SOP640_ManFrontUp
        Rectangle (715,10 160x30), "Move Up"
        Rectangle (715,60 160x30), "Upper Position"
        Rectangle (120,10 160x30), "Move Down"
        Rectangle (120,60 160x30), "Lower Position", invisible if: TRUE
        Rectangle (885,10 30x30)
            toggle SOP640_Y1
        Rectangle (80,60 30x30)
            toggle SOP640_B2
        Rectangle (80,10 30x30)
            toggle SOP640_Y2
        Rectangle (885,60 30x30)
            toggle SOP640_B3
        Polygon (991,49) (958,9) (958,89) (991,49) (991,49), invisible if: not OP60_Manual
            tap HMI_SOP640_ManFrontUp
        Polygon (9,53) (39,13) (39,93) (9,53) (9,53), invisible if: not OP60_Manual
            tap HMI_SOP640_ManFrontDown
    Group (230,600 510x68)
        Button (0,0 170x68), "SOP610t630"
            toggle OP60_Visu.CV_Manual_SOP610t630
            OnMouseDown:  Assign=Manual_SOP610t630, Type=Assignment
        Button (170,0 170x68), "SOP640"
            toggle OP60_Visu.CV_Manual_SOP640
            OnMouseDown:  Assign=Manual_SOP640, Type=Assignment
        Button (340,0 170x68), "SOP650t680"
            toggle OP60_Visu.CV_Manual_SOP650t680
            OnMouseDown:  Assign=Manual_SOP650t680, Type=Assignment
    Rectangle (10,340 1000x100), "SOP640 REAR CLAMP"
    Polygon (20,390) (50,350) (50,430) (20,390) (20,390)
    Rectangle (60,350 20x80)
        toggle HMI_SOP640_ManRearDown
    Polygon (1000,390) (967,350) (967,430) (1000,390) (1000,390)
    Rectangle (935,350 20x80)
        toggle HMI_SOP640_ManRearUp
    Rectangle (725,350 160x30), "Move Up"
    Rectangle (725,400 160x30), "Upper Position"
    Rectangle (130,350 160x30), "Move Down"
    Rectangle (130,400 160x30), "Lower Position", invisible if: TRUE
    Rectangle (895,350 30x30)
        toggle SOP640_Y3
    Rectangle (90,400 30x30)
        toggle SOP640_B4
    Rectangle (90,350 30x30)
        toggle SOP640_Y4
    Rectangle (895,400 30x30)
        toggle SOP640_B5
    Polygon (1001,389) (968,349) (968,429) (1001,389) (1001,389), invisible if: not OP60_Manual
        tap HMI_SOP640_ManRearUp
    Polygon (19,393) (49,353) (49,433) (19,393) (19,393), invisible if: not OP60_Manual
        tap HMI_SOP640_ManRearDown
    Button (780,595 232x72), "DISABLE INTERLOCKS", invisible if: not OP60_Manual
        toggle HMI_DisableInterlocks
END_VISUALIZATION

// Device/Application/Process
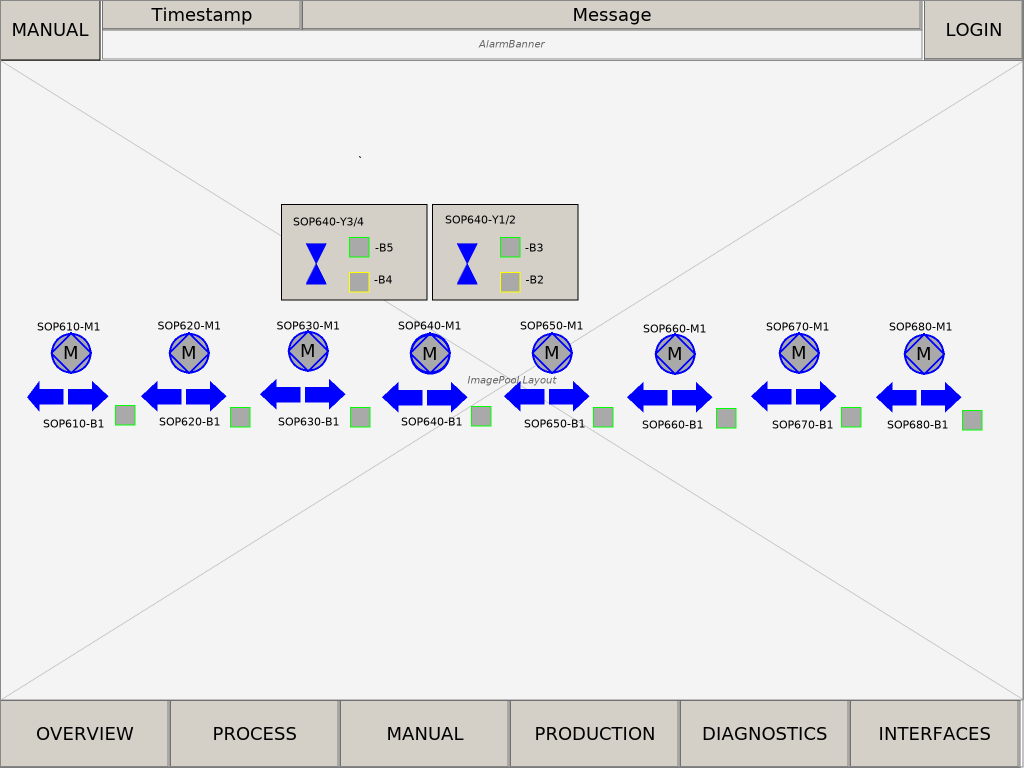
VISUALIZATION Process  // 1024x768
    Image (0,60 1024x640), image: ImagePool.Layout
    Rectangle (432,204 146x96)
    Rectangle (0,0 100x60), "AUTO"
    Rectangle (0,0 100x60), "MANUAL", invisible if: OP60_Auto
    AlarmBanner (102,29 820x30)
        p1521930926: __All
        p1663851261: __All
    Button (924,0 100x60), "LOGIN"
    Button (102,0 200x30), "Timestamp"
    Button (302,0 620x30), "Message"
    Rectangle (115,405 20x20)
        toggle SOP610_B1
    Label (22,409 104x30), "SOP610-B1"
    Ellipse (51,333 40x40), "M"
        toggle SOP610_Conveyor.oRunning
    Ellipse (51,333 40x40)
        toggle SOP610_Conveyor.oFaulted
    Polyline (51,353) (71,333) (91,353) (71,373) (51,353)
        toggle SOP610_Conveyor.oFaulted
    Rectangle (68,389 24x15), invisible if: not SOP610_Conveyor.oRunFwd and not SOP610_Conveyor.oFaulted
        toggle SOP610_Conveyor.oFaulted
    Polygon (92,388) (92,381) (108,396) (92,411) (92,403), invisible if: not SOP610_Conveyor.oRunFwd and not SOP610_Conveyor.oFaulted
        toggle SOP610_Conveyor.oFaulted
    Polygon (39,388) (39,381) (27,397) (39,411) (39,403), invisible if: not SOP610_Conveyor.oRunRev and not SOP610_Conveyor.oFaulted
        toggle SOP610_Conveyor.oFaulted
    Rectangle (39,389 24x15), invisible if: not SOP610_Conveyor.oRunRev and not SOP610_Conveyor.oFaulted
        toggle SOP610_Conveyor.oFaulted
    Label (138,407 104x30), "SOP620-B1"
    Label (257,407 104x30), "SOP630-B1"
    Label (366,407 132x30), "SOP640-B1"
    Label (503,409 104x30), "SOP650-B1"
    Label (621,410 104x30), "SOP660-B1"
    Label (866,410 104x30), "SOP680-B1"
    Label (751,410 104x30), "SOP670-B1"
    Rectangle (230,407 20x20)
        toggle SOP620_B1 p2164770859=TRUE
    Rectangle (350,407 20x20)
        toggle SOP630_B1
    Rectangle (471,406 20x20)
        toggle SOP640_B1
    Rectangle (593,407 20x20)
        toggle SOP650_B1
    Rectangle (716,408 20x20)
        toggle SOP660_B1
    Rectangle (841,407 20x20)
        toggle SOP670_B1
    Rectangle (962,410 20x20)
        toggle SOP680_B1
    Rectangle (186,389 24x15), invisible if: not SOP620_Conveyor.oRunFwd and not SOP620_Conveyor.oFaulted
        toggle SOP620_Conveyor.oFaulted
    Polygon (210,388) (210,381) (226,396) (210,411) (210,403), invisible if: not SOP620_Conveyor.oRunFwd and not SOP620_Conveyor.oFaulted
        toggle SOP620_Conveyor.oFaulted
    Ellipse (169,333 40x40), "M"
        toggle SOP620_Conveyor.oRunning
    Polygon (157,388) (157,381) (141,396) (157,411) (157,403), invisible if: not SOP620_Conveyor.oRunRev and not SOP620_Conveyor.oFaulted
        toggle SOP620_Conveyor.oFaulted
    Rectangle (157,389 24x15), invisible if: not SOP620_Conveyor.oRunRev and not SOP620_Conveyor.oFaulted
        toggle SOP620_Conveyor.oFaulted
    Rectangle (305,387 24x15), invisible if: not SOP630_Conveyor.oRunFwd and not SOP630_Conveyor.oFaulted
        toggle SOP630_Conveyor.oFaulted
    Polygon (329,386) (329,379) (345,394) (329,409) (329,401), invisible if: not SOP630_Conveyor.oRunFwd and not SOP630_Conveyor.oFaulted
        toggle SOP630_Conveyor.oFaulted
    Ellipse (288,331 40x40), "M"
        toggle SOP630_Conveyor.oRunning
    Polygon (276,386) (276,379) (260,394) (276,409) (276,401), invisible if: not SOP630_Conveyor.oRunRev and not SOP630_Conveyor.oFaulted
        toggle SOP630_Conveyor.oFaulted
    Rectangle (276,387 24x15), invisible if: not SOP630_Conveyor.oRunRev and not SOP630_Conveyor.oFaulted
        toggle SOP630_Conveyor.oFaulted
    Rectangle (427,390 24x15), invisible if: not SOP640_Conveyor.oRunFwd and not SOP640_Conveyor.oFaulted
        toggle SOP640_Conveyor.oFaulted
    Polygon (451,389) (451,382) (467,397) (451,412) (451,404), invisible if: not SOP640_Conveyor.oRunFwd and not SOP640_Conveyor.oFaulted
        toggle SOP640_Conveyor.oFaulted
    Ellipse (410,334 40x40), "M"
        toggle SOP640_Conveyor.oRunning
    Polygon (398,389) (398,382) (382,397) (398,412) (398,404), invisible if: not SOP640_Conveyor.oRunRev and not SOP640_Conveyor.oFaulted
        toggle SOP640_Conveyor.oFaulted
    Rectangle (398,390 24x15), invisible if: not SOP640_Conveyor.oRunRev and not SOP640_Conveyor.oFaulted
        toggle SOP640_Conveyor.oFaulted
    Rectangle (549,389 24x15), invisible if: not SOP650_Conveyor.oRunFwd and not SOP650_Conveyor.oFaulted
        toggle SOP650_Conveyor.oFaulted
    Polygon (573,388) (573,381) (589,396) (573,411) (573,403), invisible if: not SOP650_Conveyor.oRunFwd and not SOP650_Conveyor.oFaulted
        toggle SOP650_Conveyor.oFaulted
    Ellipse (532,333 40x40), "M"
        toggle SOP650_Conveyor.oRunning
    Polygon (520,388) (520,381) (504,396) (520,411) (520,403), invisible if: not SOP650_Conveyor.oRunRev and not SOP650_Conveyor.oFaulted
        toggle SOP650_Conveyor.oFaulted
    Rectangle (520,389 24x15), invisible if: not SOP650_Conveyor.oRunRev and not SOP650_Conveyor.oFaulted
        toggle SOP650_Conveyor.oFaulted
    Rectangle (672,390 24x15), invisible if: not SOP660_Conveyor.oRunFwd and not SOP660_Conveyor.oFaulted
        toggle SOP660_Conveyor.oFaulted
    Polygon (696,389) (696,382) (712,397) (696,412) (696,404), invisible if: not SOP660_Conveyor.oRunFwd and not SOP660_Conveyor.oFaulted
        toggle SOP660_Conveyor.oFaulted
    Ellipse (655,334 40x40), "M"
        toggle SOP660_Conveyor.oRunning
    Polygon (643,389) (643,382) (627,397) (643,412) (643,404), invisible if: not SOP660_Conveyor.oRunRev and not SOP660_Conveyor.oFaulted
        toggle SOP660_Conveyor.oFaulted
    Rectangle (643,390 24x15), invisible if: not SOP660_Conveyor.oRunRev and not SOP660_Conveyor.oFaulted
        toggle SOP660_Conveyor.oFaulted
    Rectangle (796,389 24x15), invisible if: not SOP670_Conveyor.oRunFwd and not SOP670_Conveyor.oFaulted
        toggle SOP670_Conveyor.oFaulted
    Polygon (820,388) (820,381) (836,396) (820,411) (820,403), invisible if: not SOP670_Conveyor.oRunFwd and not SOP670_Conveyor.oFaulted
        toggle SOP670_Conveyor.oFaulted
    Ellipse (779,333 40x40), "M"
        toggle SOP670_Conveyor.oRunning
    Polygon (767,388) (767,381) (751,396) (767,411) (767,403), invisible if: not SOP670_Conveyor.oRunRev and not SOP670_Conveyor.oFaulted
        toggle SOP670_Conveyor.oFaulted
    Rectangle (767,389 24x15), invisible if: not SOP670_Conveyor.oRunRev and not SOP670_Conveyor.oFaulted
        toggle SOP670_Conveyor.oFaulted
    Rectangle (921,390 24x15), invisible if: not SOP680_Conveyor.oRunFwd and not SOP680_Conveyor.oFaulted
        toggle SOP680_Conveyor.oFaulted
    Polygon (945,389) (945,382) (961,397) (945,412) (945,404), invisible if: not SOP680_Conveyor.oRunFwd and not SOP680_Conveyor.oFaulted
        toggle SOP680_Conveyor.oFaulted
    Ellipse (904,334 40x40), "M"
        toggle SOP680_Conveyor.oRunning
    Polygon (892,389) (892,382) (876,397) (892,412) (892,404), invisible if: not SOP680_Conveyor.oRunRev and not SOP680_Conveyor.oFaulted
        toggle SOP680_Conveyor.oFaulted
    Rectangle (892,390 24x15), invisible if: not SOP680_Conveyor.oRunRev and not SOP680_Conveyor.oFaulted
        toggle SOP680_Conveyor.oFaulted
    Ellipse (169,333 40x40)
        toggle SOP620_Conveyor.oFaulted
    Polyline (169,353) (189,333) (209,353) (189,373) (169,353)
        toggle SOP620_Conveyor.oFaulted
    Ellipse (288,331 40x40)
        toggle SOP630_Conveyor.oFaulted
    Polyline (288,351) (308,331) (328,351) (308,371) (288,351)
        toggle SOP630_Conveyor.oFaulted
    Ellipse (410,333 40x40)
        toggle SOP640_Conveyor.oFaulted
    Polyline (410,353) (430,333) (450,353) (430,373) (410,353)
        toggle SOP640_Conveyor.oFaulted
    Ellipse (532,333 40x40)
        toggle SOP650_Conveyor.oFaulted
    Polyline (532,353) (552,333) (572,353) (552,373) (532,353)
        toggle SOP650_Conveyor.oFaulted
    Ellipse (655,334 40x40)
        toggle SOP660_Conveyor.oFaulted
    Polyline (655,354) (675,334) (695,354) (675,374) (655,354)
        toggle SOP660_Conveyor.oFaulted
    Ellipse (779,333 40x40)
        toggle SOP670_Conveyor.oFaulted
    Polyline (779,353) (799,333) (819,353) (799,373) (779,353)
        toggle SOP670_Conveyor.oFaulted
    Ellipse (904,334 40x40)
        toggle SOP680_Conveyor.oFaulted
    Polyline (904,354) (924,334) (944,354) (924,374) (904,354)
        toggle SOP680_Conveyor.oFaulted
    Polygon (359,156) (360,157)
    Polygon (457,243) (477,243) (467,263) (457,283) (477,283)
    Polygon (457,244) (477,244) (467,264) (457,284) (477,284), invisible if: not SOP640_Conveyor.oFrontClampDown and not SOP640_Conveyor.oFrontClampUp and not SOP640_Conveyor.oFaulted
        toggle SOP640_Conveyor.oFaulted
    Rectangle (500,237 20x20)
        toggle SOP640_B3
    Rectangle (500,272 20x20)
        toggle SOP640_B2
    Label (415,205 131x30), "SOP640-Y1/2"
    Label (508,233 53x30), "-B3"
    Label (509,265 52x30), "-B2"
    Rectangle (281,204 146x96)
    Polygon (306,243) (326,243) (316,263) (306,283) (326,283)
    Polygon (306,244) (326,244) (316,264) (306,284) (326,284), invisible if: not SOP640_Conveyor.oRearClampDown and not SOP640_Conveyor.oRearClampUp and not SOP640_Conveyor.oFaulted
        toggle SOP640_Conveyor.oFaulted
    Rectangle (349,237 20x20)
        toggle SOP640_B5
    Rectangle (349,272 20x20)
        toggle SOP640_B4
    Label (263,207 131x30), "SOP640-Y3/4"
    Label (358,233 53x30), "-B5"
    Label (358,265 51x30), "-B4"
    Group (0,700 1020x68)
        Button (0,0 170x68), "OVERVIEW"
            toggle OP60_Visu.CV_Overview
            OnMouseDown:  Assign=Overview, Type=Assignment
        Button (170,0 170x68), "PROCESS"
            toggle OP60_Visu.CV_Process
            OnMouseDown:  Assign=Process, Type=Assignment
        Button (340,0 170x68), "MANUAL"
            toggle OP60_Visu.CV_Manual_SOP610t630
            OnMouseDown:  Assign=Manual_SOP610t630, Type=Assignment
        Button (510,0 170x68), "PRODUCTION"
            toggle OP60_Visu.CV_Production
            OnMouseDown:  Assign=Production, Type=Assignment
        Button (680,0 170x68), "DIAGNOSTICS"
            toggle OP60_Visu.CV_Diagnostics
            OnMouseDown:  Assign=Diagnostics, Type=Assignment
        Button (850,0 170x68), "INTERFACES"
            toggle OP60_Visu.CV_Interfaces
            OnMouseDown:  Assign=Interfaces, Type=Assignment
    Label (28,312 82x30), "SOP610-M1"
    Label (142,311 95x30), "SOP620-M1"
    Label (265,311 87x30), "SOP630-M1"
    Label (386,311 88x30), "SOP640-M1"
    Label (508,311 88x30), "SOP650-M1"
    Label (631,314 88x30), "SOP660-M1"
    Label (754,312 88x30), "SOP670-M1"
    Label (877,312 88x30), "SOP680-M1"
END_VISUALIZATION

// Device/Application/Interfaces
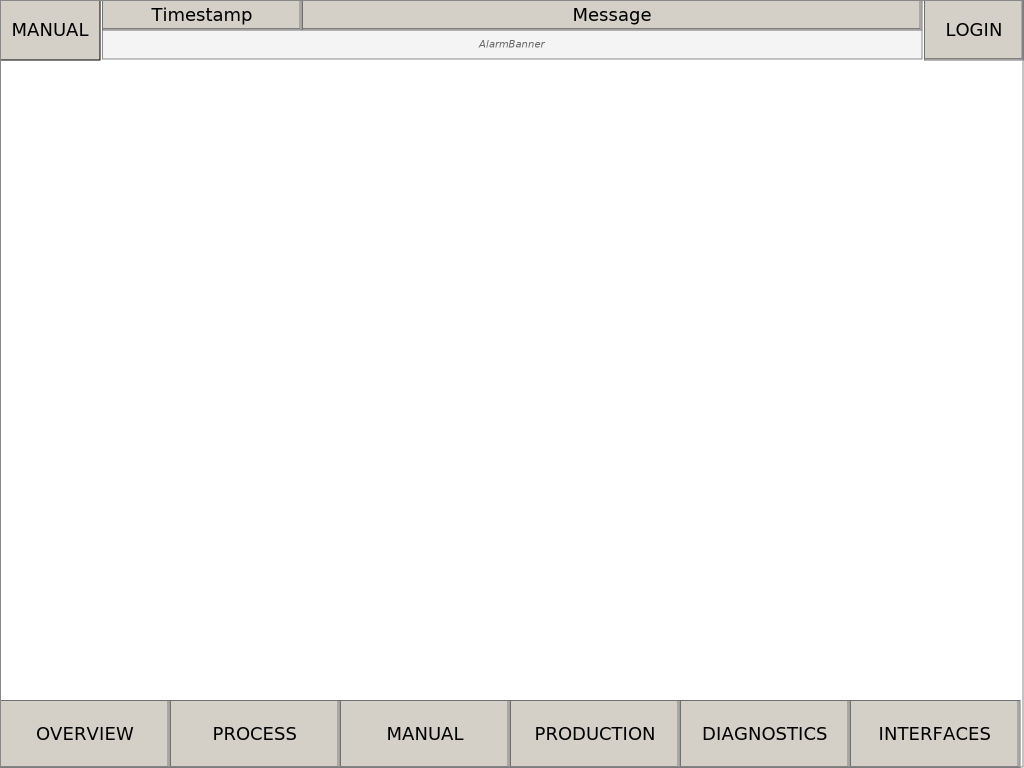
VISUALIZATION Interfaces  // 1024x768
    Rectangle (0,0 100x60), "AUTO"
    Rectangle (0,0 100x60), "MANUAL", invisible if: OP60_Auto
    AlarmBanner (102,29 820x30)
        p1521930926: __All
        p1663851261: __All
    Button (924,0 100x60), "LOGIN"
    Button (102,0 200x30), "Timestamp"
    Button (302,0 620x30), "Message"
    Group (0,700 1020x68)
        Button (0,0 170x68), "OVERVIEW"
            toggle OP60_Visu.CV_Overview
            OnMouseDown:  Assign=Overview, Type=Assignment
        Button (170,0 170x68), "PROCESS"
            toggle OP60_Visu.CV_Process
            OnMouseDown:  Assign=Process, Type=Assignment
        Button (340,0 170x68), "MANUAL"
            toggle OP60_Visu.CV_Manual_SOP610t630
            OnMouseDown:  Assign=Manual_SOP610t630, Type=Assignment
        Button (510,0 170x68), "PRODUCTION"
            toggle OP60_Visu.CV_Production
            OnMouseDown:  Assign=Production, Type=Assignment
        Button (680,0 170x68), "DIAGNOSTICS"
            toggle OP60_Visu.CV_Diagnostics
            OnMouseDown:  Assign=Diagnostics, Type=Assignment
        Button (850,0 170x68), "INTERFACES"
            toggle OP60_Visu.CV_Interfaces
            OnMouseDown:  Assign=Interfaces, Type=Assignment
END_VISUALIZATION

// /Production
VISUALIZATION Production  // 1024x768
END_VISUALIZATION

// Device/Application/Diagnostics
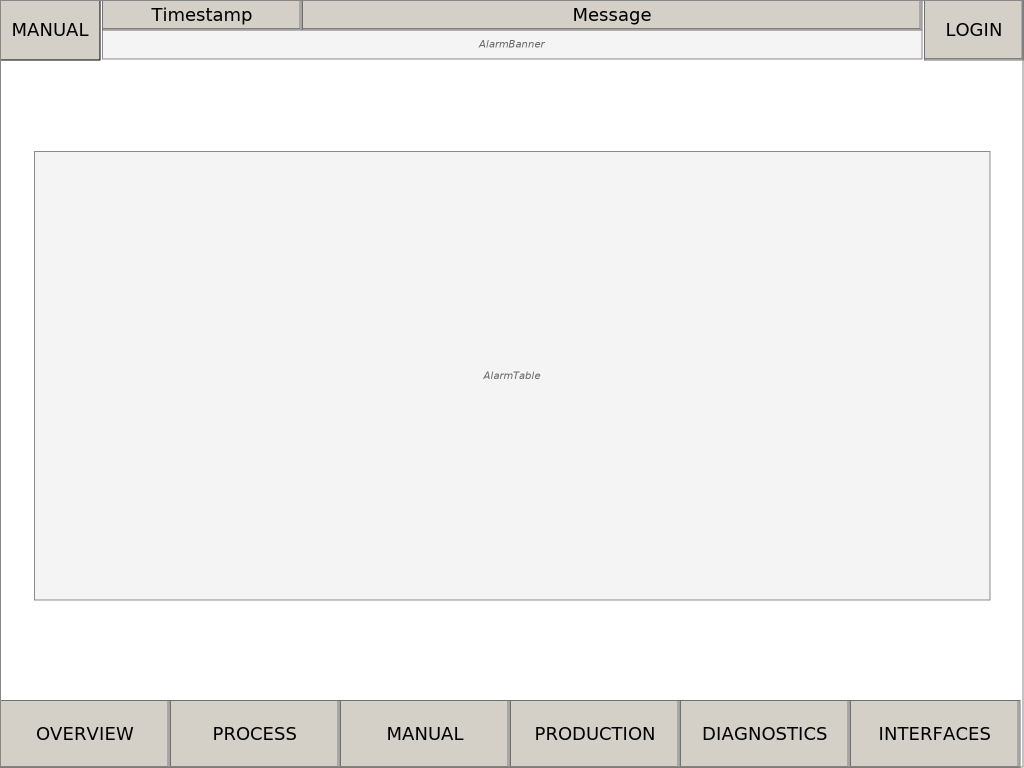
VISUALIZATION Diagnostics  // 1024x768
    Group (0,700 1020x68)
        Button (0,0 170x68), "OVERVIEW"
            toggle OP60_Visu.CV_Overview
            OnMouseDown:  Assign=Overview, Type=Assignment
        Button (170,0 170x68), "PROCESS"
            toggle OP60_Visu.CV_Process
            OnMouseDown:  Assign=Process, Type=Assignment
        Button (340,0 170x68), "MANUAL"
            toggle OP60_Visu.CV_Manual_SOP610t630
            OnMouseDown:  Assign=Manual_SOP610t630, Type=Assignment
        Button (510,0 170x68), "PRODUCTION"
            toggle OP60_Visu.CV_Production
            OnMouseDown:  Assign=Production, Type=Assignment
        Button (680,0 170x68), "DIAGNOSTICS"
            toggle OP60_Visu.CV_Diagnostics
            OnMouseDown:  Assign=Diagnostics, Type=Assignment
        Button (850,0 170x68), "INTERFACES"
            toggle OP60_Visu.CV_Interfaces
            OnMouseDown:  Assign=Interfaces, Type=Assignment
    Rectangle (0,0 100x60), "AUTO"
    Rectangle (0,0 100x60), "MANUAL", invisible if: OP60_Auto
    AlarmBanner (102,29 820x30)
        p1521930926: __All
        p1663851261: __All
    Button (924,0 100x60), "LOGIN"
    Button (102,0 200x30), "Timestamp"
    Button (302,0 620x30), "Message"
    AlarmTable (34,151 956x449)
        p1521930926: __All
        p1663851261: __All
END_VISUALIZATION

// Device/Application/Manual_SOP610t630
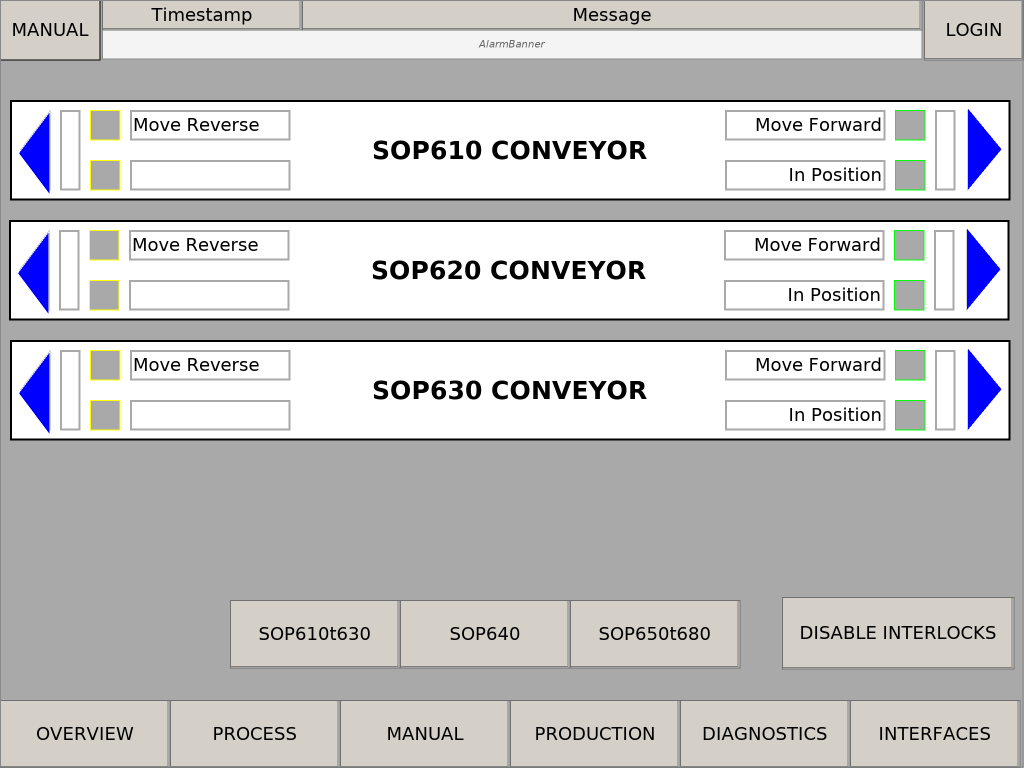
VISUALIZATION Manual_SOP610t630  // 1024x768
    Rectangle (0,0 100x60), "AUTO"
    Rectangle (0,0 100x60), "MANUAL", invisible if: OP60_Auto
    AlarmBanner (102,29 820x30)
        p1521930926: __All
        p1663851261: __All
    Button (924,0 100x60), "LOGIN"
    Button (102,0 200x30), "Timestamp"
    Button (302,0 620x30), "Message"
    Group (230,600 510x68)
        Button (0,0 170x68), "SOP610t630"
            toggle OP60_Visu.CV_Manual_SOP610t630
            OnMouseDown:  Assign=Manual_SOP610t630, Type=Assignment
        Button (170,0 170x68), "SOP640"
            toggle OP60_Visu.CV_Manual_SOP640
            OnMouseDown:  Assign=Manual_SOP640, Type=Assignment
        Button (340,0 170x68), "SOP650t680"
            toggle OP60_Visu.CV_Manual_SOP650t680
            OnMouseDown:  Assign=Manual_SOP650t680, Type=Assignment
    Button (0,700 170x68), "OVERVIEW"
        toggle OP60_Visu.CV_Overview
        OnMouseDown:  Assign=Overview, Type=Assignment
    Button (170,700 170x68), "PROCESS"
        toggle OP60_Visu.CV_Process
        OnMouseDown:  Assign=Process, Type=Assignment
    Button (340,700 170x68), "MANUAL"
        toggle OP60_Visu.CV_Manual_SOP610t630
        OnMouseDown:  Assign=Manual_SOP610t630, Type=Assignment
    Button (510,700 170x68), "PRODUCTION"
        toggle OP60_Visu.CV_Production
        OnMouseDown:  Assign=Production, Type=Assignment
    Button (680,700 170x68), "DIAGNOSTICS"
        toggle OP60_Visu.CV_Diagnostics
        OnMouseDown:  Assign=Diagnostics, Type=Assignment
    Button (850,700 170x68), "INTERFACES"
        toggle OP60_Visu.CV_Interfaces
        OnMouseDown:  Assign=Interfaces, Type=Assignment
    Rectangle (10,100 1000x100), "SOP610 CONVEYOR"
    Polygon (20,150) (50,110) (50,190) (20,150) (20,150)
    Rectangle (60,110 20x80)
        toggle HMI_SOP610_ManMoveRev
    Polygon (1000,150) (967,110) (967,190) (1000,150) (1000,150)
    Rectangle (935,110 20x80)
        toggle HMI_SOP610_ManMoveFwd
    Rectangle (725,110 160x30), "Move Forward"
    Rectangle (725,160 160x30), "In Position"
    Rectangle (130,110 160x30), "Move Reverse"
    Rectangle (130,160 160x30), invisible if: TRUE
    Rectangle (895,110 30x30)
        toggle SOP610_KM1
    Rectangle (90,160 30x30), invisible if: TRUE
    Rectangle (90,110 30x30)
        toggle SOP610_KM2
    Rectangle (895,160 30x30)
        toggle SOP610_B1
    Polygon (1001,149) (968,109) (968,189) (1001,149) (1001,149), invisible if: not OP60_Manual
        tap HMI_SOP610_ManMoveFwd
    Polygon (19,153) (49,113) (49,193) (19,153) (19,153), invisible if: not OP60_Manual
        tap HMI_SOP610_ManMoveRev
    Group (9,220 1000x100)
        Rectangle (0,0 1000x100), "SOP620 CONVEYOR"
        Polygon (10,50) (40,10) (40,90) (10,50) (10,50)
        Rectangle (50,10 20x80)
            toggle HMI_SOP620_ManMoveRev
        Polygon (990,50) (957,10) (957,90) (990,50) (990,50)
        Rectangle (925,10 20x80)
            toggle HMI_SOP620_ManMoveFwd
        Rectangle (715,10 160x30), "Move Forward"
        Rectangle (715,60 160x30), "In Position"
        Rectangle (120,10 160x30), "Move Reverse"
        Rectangle (120,60 160x30), invisible if: TRUE
        Rectangle (885,10 30x30)
            toggle SOP620_KM1
        Rectangle (80,60 30x30), invisible if: TRUE
        Rectangle (80,10 30x30)
            toggle SOP620_KM2
        Rectangle (885,60 30x30)
            toggle SOP620_B1
        Polygon (991,49) (958,9) (958,89) (991,49) (991,49), invisible if: not OP60_Manual
            tap HMI_SOP620_ManMoveFwd
        Polygon (9,53) (39,13) (39,93) (9,53) (9,53), invisible if: not OP60_Manual
            tap HMI_SOP620_ManMoveRev
    Group (10,340 1000x100)
        Rectangle (0,0 1000x100), "SOP630 CONVEYOR"
        Polygon (10,50) (40,10) (40,90) (10,50) (10,50)
        Rectangle (50,10 20x80)
            toggle HMI_SOP630_ManMoveRev
        Polygon (990,50) (957,10) (957,90) (990,50) (990,50)
        Rectangle (925,10 20x80)
            toggle HMI_SOP630_ManMoveFwd
        Rectangle (715,10 160x30), "Move Forward"
        Rectangle (715,60 160x30), "In Position"
        Rectangle (120,10 160x30), "Move Reverse"
        Rectangle (120,60 160x30), invisible if: TRUE
        Rectangle (885,10 30x30)
            toggle SOP630_KM1
        Rectangle (80,60 30x30), invisible if: TRUE
        Rectangle (80,10 30x30)
            toggle SOP630_KM2
        Rectangle (885,60 30x30)
            toggle SOP630_B1
        Polygon (991,49) (958,9) (958,89) (991,49) (991,49), invisible if: not OP60_Manual
            tap HMI_SOP630_ManMoveFwd
        Polygon (9,53) (39,13) (39,93) (9,53) (9,53), invisible if: not OP60_Manual
            tap HMI_SOP630_ManMoveRev
    Button (782,597 232x72), "DISABLE INTERLOCKS", invisible if: not OP60_Manual
        toggle HMI_DisableInterlocks
END_VISUALIZATION

// Device/Application/Manual_SOP650t680
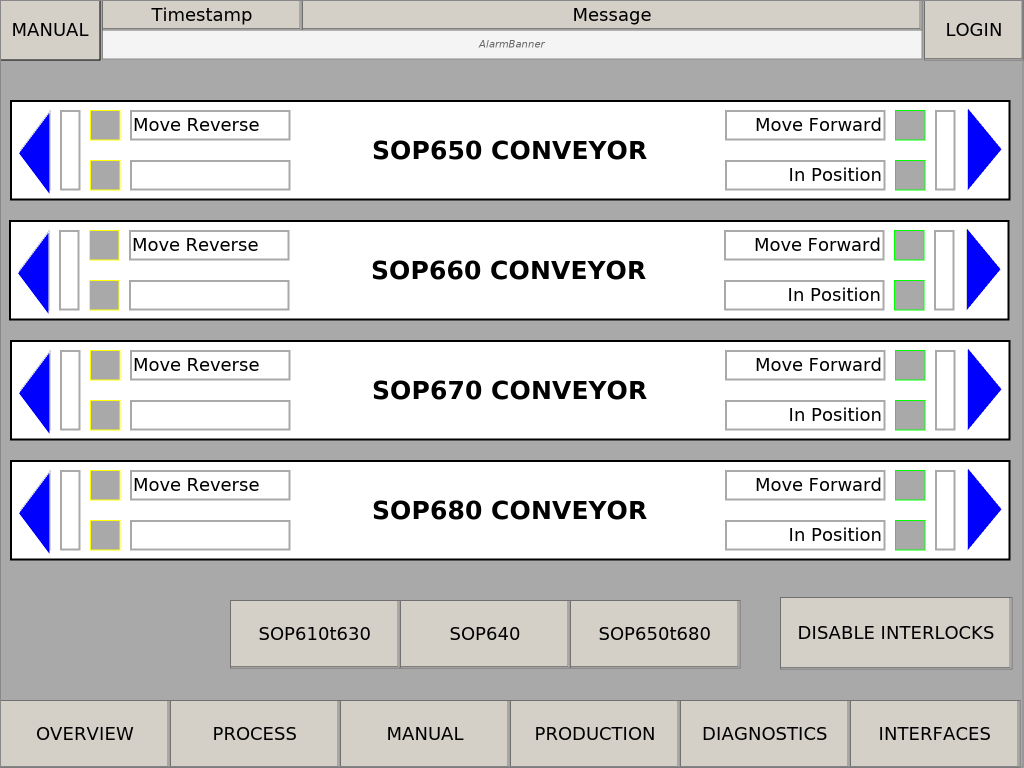
VISUALIZATION Manual_SOP650t680  // 1024x768
    Rectangle (0,0 100x60), "AUTO"
    Rectangle (0,0 100x60), "MANUAL", invisible if: OP60_Auto
    AlarmBanner (102,29 820x30)
        p1521930926: __All
        p1663851261: __All
    Button (924,0 100x60), "LOGIN"
    Button (102,0 200x30), "Timestamp"
    Button (302,0 620x30), "Message"
    Button (0,700 170x68), "OVERVIEW"
        toggle OP60_Visu.CV_Overview
        OnMouseDown:  Assign=Overview, Type=Assignment
    Button (170,700 170x68), "PROCESS"
        toggle OP60_Visu.CV_Process
        OnMouseDown:  Assign=Process, Type=Assignment
    Button (340,700 170x68), "MANUAL"
        toggle OP60_Visu.CV_Manual_SOP610t630
        OnMouseDown:  Assign=Manual_SOP610t630, Type=Assignment
    Button (510,700 170x68), "PRODUCTION"
        toggle OP60_Visu.CV_Production
        OnMouseDown:  Assign=Production, Type=Assignment
    Button (680,700 170x68), "DIAGNOSTICS"
        toggle OP60_Visu.CV_Diagnostics
        OnMouseDown:  Assign=Diagnostics, Type=Assignment
    Button (850,700 170x68), "INTERFACES"
        toggle OP60_Visu.CV_Interfaces
        OnMouseDown:  Assign=Interfaces, Type=Assignment
    Group (10,100 1000x100)
        Rectangle (0,0 1000x100), "SOP650 CONVEYOR"
        Polygon (10,50) (40,10) (40,90) (10,50) (10,50)
        Rectangle (50,10 20x80)
            toggle HMI_SOP650_ManMoveRev
        Polygon (990,50) (957,10) (957,90) (990,50) (990,50)
        Rectangle (925,10 20x80)
            toggle HMI_SOP650_ManMoveFwd
        Rectangle (715,10 160x30), "Move Forward"
        Rectangle (715,60 160x30), "In Position"
        Rectangle (120,10 160x30), "Move Reverse"
        Rectangle (120,60 160x30), invisible if: TRUE
        Rectangle (885,10 30x30)
            toggle SOP650_KM1
        Rectangle (80,60 30x30), invisible if: TRUE
        Rectangle (80,10 30x30)
            toggle SOP650_KM2
        Rectangle (885,60 30x30)
            toggle SOP650_B1
        Polygon (991,49) (958,9) (958,89) (991,49) (991,49), invisible if: not OP60_Manual
            tap HMI_SOP650_ManMoveFwd
        Polygon (9,53) (39,13) (39,93) (9,53) (9,53), invisible if: not OP60_Manual
            tap HMI_SOP650_ManMoveRev
    Group (9,220 1000x100)
        Rectangle (0,0 1000x100), "SOP660 CONVEYOR"
        Polygon (10,50) (40,10) (40,90) (10,50) (10,50)
        Rectangle (50,10 20x80)
            toggle HMI_SOP660_ManMoveRev
        Polygon (990,50) (957,10) (957,90) (990,50) (990,50)
        Rectangle (925,10 20x80)
            toggle HMI_SOP660_ManMoveFwd
        Rectangle (715,10 160x30), "Move Forward"
        Rectangle (715,60 160x30), "In Position"
        Rectangle (120,10 160x30), "Move Reverse"
        Rectangle (120,60 160x30), invisible if: TRUE
        Rectangle (885,10 30x30)
            toggle SOP660_KM1
        Rectangle (80,60 30x30), invisible if: TRUE
        Rectangle (80,10 30x30)
            toggle SOP660_KM2
        Rectangle (885,60 30x30)
            toggle SOP660_B1
        Polygon (991,49) (958,9) (958,89) (991,49) (991,49), invisible if: not OP60_Manual
            tap HMI_SOP660_ManMoveFwd
        Polygon (9,53) (39,13) (39,93) (9,53) (9,53), invisible if: not OP60_Manual
            tap HMI_SOP660_ManMoveRev
    Group (10,340 1000x100)
        Rectangle (0,0 1000x100), "SOP670 CONVEYOR"
        Polygon (10,50) (40,10) (40,90) (10,50) (10,50)
        Rectangle (50,10 20x80)
            toggle HMI_SOP670_ManMoveRev
        Polygon (990,50) (957,10) (957,90) (990,50) (990,50)
        Rectangle (925,10 20x80)
            toggle HMI_SOP670_ManMoveFwd
        Rectangle (715,10 160x30), "Move Forward"
        Rectangle (715,60 160x30), "In Position"
        Rectangle (120,10 160x30), "Move Reverse"
        Rectangle (120,60 160x30), invisible if: TRUE
        Rectangle (885,10 30x30)
            toggle SOP670_KM1
        Rectangle (80,60 30x30), invisible if: TRUE
        Rectangle (80,10 30x30)
            toggle SOP670_KM2
        Rectangle (885,60 30x30)
            toggle SOP670_B1
        Polygon (991,49) (958,9) (958,89) (991,49) (991,49), invisible if: not OP60_Manual
            tap HMI_SOP670_ManMoveFwd
        Polygon (9,53) (39,13) (39,93) (9,53) (9,53), invisible if: not OP60_Manual
            tap HMI_SOP670_ManMoveRev
    Group (10,460 1000x100)
        Rectangle (0,0 1000x100), "SOP680 CONVEYOR"
        Polygon (10,50) (40,10) (40,90) (10,50) (10,50)
        Rectangle (50,10 20x80)
            toggle HMI_SOP680_ManMoveRev
        Polygon (990,50) (957,10) (957,90) (990,50) (990,50)
        Rectangle (925,10 20x80)
            toggle HMI_SOP680_ManMoveFwd
        Rectangle (715,10 160x30), "Move Forward"
        Rectangle (715,60 160x30), "In Position"
        Rectangle (120,10 160x30), "Move Reverse"
        Rectangle (120,60 160x30), invisible if: TRUE
        Rectangle (885,10 30x30)
            toggle SOP680_KM1
        Rectangle (80,60 30x30), invisible if: TRUE
        Rectangle (80,10 30x30)
            toggle SOP680_KM2
        Rectangle (885,60 30x30)
            toggle SOP680_B1
        Polygon (991,49) (958,9) (958,89) (991,49) (991,49), invisible if: not OP60_Manual
            tap HMI_SOP680_ManMoveFwd
        Polygon (9,53) (39,13) (39,93) (9,53) (9,53), invisible if: not OP60_Manual
            tap HMI_SOP680_ManMoveRev
    Group (230,600 510x68)
        Button (0,0 170x68), "SOP610t630"
            toggle OP60_Visu.CV_Manual_SOP610t630
            OnMouseDown:  Assign=Manual_SOP610t630, Type=Assignment
        Button (170,0 170x68), "SOP640"
            toggle OP60_Visu.CV_Manual_SOP640
            OnMouseDown:  Assign=Manual_SOP640, Type=Assignment
        Button (340,0 170x68), "SOP650t680"
            toggle OP60_Visu.CV_Manual_SOP650t680
            OnMouseDown:  Assign=Manual_SOP650t680, Type=Assignment
    Button (780,597 232x72), "DISABLE INTERLOCKS", invisible if: not OP60_Manual
        toggle HMI_DisableInterlocks
END_VISUALIZATION

(* text list TextList (id | default)
  6813 | SOP680 Conveyor PD Mismatch, has a product but not a valid PD
  6814 | SOP680 Conveyor PD Mismatch, has no product but PD is not empty
  6713 | SOP670 Conveyor PD Mismatch, has a product but not a valid PD
  6714 | SOP670 Conveyor PD Mismatch, has no product but PD is not empty
  6613 | SOP660 Conveyor PD Mismatch, has a product but not a valid PD
  6614 | SOP660 Conveyor PD Mismatch, has no product but PD is not empty
  6513 | SOP650 Conveyor PD Mismatch, has a product but not a valid PD
  6514 | SOP650 Conveyor PD Mismatch, has no product but PD is not empty
  6413 | SOP640 Conveyor PD Mismatch, has a product but not a valid PD
  6414 | SOP640 Conveyor PD Mismatch, has no product but PD is not empty
  6313 | SOP630 Conveyor PD Mismatch, has a product but not a valid PD
  6314 | SOP630 Conveyor PD Mismatch, has no product but PD is not empty
  6213 | SOP620 Conveyor PD Mismatch, has a product but not a valid PD
  6214 | SOP620 Conveyor PD Mismatch, has no product but PD is not empty
  6114 | SOP610 Conveyor PD Mismatch, has no product but PD is not empty
  6113 | SOP610 Conveyor PD Mismatch, has a product but not a valid PD
  6423 | SOP640: Rear Clamp Pair Check Fault
  6422 | SOP640: Front Clamp Pair Check Fault
  6421 | SOP640: Timeout Rear Clamp
  6420 | SOP640: Timeout Front Clamp
  6008 | SOP040_B1: Pneumatic Pressure is not OK
  0603 | OP60 Manual Interlocks Disabled
  6430 | SOP640-LC1: Light Curtain has been cut
  6902 | SOP690-B1: Safety Door Open
  6901 | SOP690-NS1: Emergency Stop
  6007 | SOP600-NS1: Emergency Stop
  6006 | SOP024-F13: Safety Circuit Protection
  6005 | SOP024-F12: PLC Output Protection
  6004 | SOP024-F11: PLC Input Protection
  6003 | SOP024-F10: Power Supply Sec. Protection
  6002 | SOP024-FQ1: Power Supply Prim. Protection
  0602 | OP60 in Empty Mode
  6001 | SOP010_FQ1: Power Line Circuit Breaker
  0601 | OP60 Waiting to OP50
  6111 | SOP610 Conveyor PD Transfer Error, previous Conveyor has no PD
  6205 | SOP620 Conveyor Motor Protection Tripped
  6106 | SOP610 Conveyor Motor Protection Tripped
  6105 | SOP610 Conveyor Motor Protection Tripped
  6102 | SOP610 Conveyor Timeout Transfering
  6101 | SOP610 Conveyor Timeout Loading
  6110 | SOP610 Conveyor PD Transfer Error, next Conveyor has PD
  6112 | SOP610 Conveyor PD Transfer Error, Conveyor has no PD
  6202 | SOP620 Conveyor Timeout Transfering
  6201 | SOP620 Conveyor Timeout Loading
  6210 | SOP620 Conveyor PD Transfer Error, next Conveyor has PD
  6211 | SOP620 Conveyor PD Transfer Error, previous Conveyor has no PD
  6212 | SOP620 Conveyor PD Transfer Error, Conveyor has no PD
  6301 | SOP630 Conveyor Timeout Loading
  6302 | SOP630 Conveyor Timeout Transfering
  6305 | SOP630 Conveyor Motor Protection Tripped
  6310 | SOP630 Conveyor PD Transfer Error, next Conveyor has PD
  6311 | SOP630 Conveyor PD Transfer Error, previous Conveyor has no PD
  6312 | SOP630 Conveyor PD Transfer Error, Conveyor has no PD
  6401 | SOP640 Conveyor Timeout Loading
  6402 | SOP640 Conveyor Timeout Transfering
  6405 | SOP640 Conveyor Motor Protection Tripped
  6410 | SOP640 Conveyor PD Transfer Error, next Conveyor has PD
  6411 | SOP640 Conveyor PD Transfer Error, previous Conveyor has no PD
  6412 | SOP640 Conveyor PD Transfer Error, Conveyor has no PD
  6501 | SOP650 Conveyor Timeout Loading
  6502 | SOP650 Conveyor Timeout Transfering
  6505 | SOP650 Conveyor Motor Protection Tripped
  6510 | SOP650 Conveyor PD Transfer Error, next Conveyor has PD
  6511 | SOP650 Conveyor PD Transfer Error, previous Conveyor has no PD
  6512 | SOP650 Conveyor PD Transfer Error, Conveyor has no PD
  6601 | SOP660 Conveyor Timeout Loading
  6602 | SOP660 Conveyor Timeout Transfering
  6605 | SOP660 Conveyor Motor Protection Tripped
  6610 | SOP660 Conveyor PD Transfer Error, next Conveyor has PD
  6611 | SOP660 Conveyor PD Transfer Error, previous Conveyor has no PD
  6612 | SOP660 Conveyor PD Transfer Error, Conveyor has no PD
  6701 | SOP670 Conveyor Timeout Loading
  6702 | SOP670 Conveyor Timeout Transfering
  6705 | SOP670 Conveyor Motor Protection Tripped
  6710 | SOP670 Conveyor PD Transfer Error, next Conveyor has PD
  6711 | SOP670 Conveyor PD Transfer Error, previous Conveyor has no PD
  6712 | SOP670 Conveyor PD Transfer Error, Conveyor has no PD
  6801 | SOP680 Conveyor Timeout Loading
  6802 | SOP680 Conveyor Timeout Transfering
  6805 | SOP680 Conveyor Motor Protection Tripped
  6810 | SOP680 Conveyor PD Transfer Error, next Conveyor has PD
  6811 | SOP680 Conveyor PD Transfer Error, previous Conveyor has no PD
  6812 | SOP680 Conveyor PD Transfer Error, Conveyor has no PD
   |  *)

(* text list System (id | default)
  Apr | Apr
  April | April
  Aug | Aug
  August | August
  Dec | Dec
  December | December
  Feb | Feb
  February | February
  Fri | Fri
  Friday | Friday
  Jan | Jan
  January | January
  Jul | Jul
  July | July
  Jun | Jun
  June | June
  Mar | Mar
  March | March
  May | May
  May_3Letter | May
  Mon | Mon
  Monday | Monday
  Nov | Nov
  November | November
  Oct | Oct
  October | October
  Sat | Sat
  Saturday | Saturday
  Sep | Sep
  September | September
  Sun | Sun
  Sunday | Sunday
  Thu | Thu
  Thursday | Thursday
  Tue | Tue
  Tuesday | Tuesday
  Wed | Wed
  Wednesday | Wednesday
   |  *)
